(* IEC 61131-3 sources: TA/Tests/RetainTest/Man (part 6) *)

    RETAINTEST_AUTO_ARRAYARRAY_TIME[1][0] := RETAINTEST_AUTO_ARRAYARRAY_TIME[1][0] + PULSE_TIME;
    RETAINTEST_AUTO_ARRAYARRAY_TIME[1][1] := RETAINTEST_AUTO_ARRAYARRAY_TIME[1][1] + PULSE_TIME;
    RETAINTEST_AUTO_ARRAYARRAY_TIME[1][2] := RETAINTEST_AUTO_ARRAYARRAY_TIME[1][2] + PULSE_TIME;
    RETAINTEST_AUTO_ARRAYARRAY_TIME[1][3] := RETAINTEST_AUTO_ARRAYARRAY_TIME[1][3] + PULSE_TIME;
    RETAINTEST_AUTO_ARRAYARRAY_TIME[1][4] := RETAINTEST_AUTO_ARRAYARRAY_TIME[1][4] + PULSE_TIME;
    RETAINTEST_AUTO_ARRAYARRAY_TIME[1][5] := RETAINTEST_AUTO_ARRAYARRAY_TIME[1][5] + PULSE_TIME;
    RETAINTEST_AUTO_ARRAYARRAY_TIME[1][6] := RETAINTEST_AUTO_ARRAYARRAY_TIME[1][6] + PULSE_TIME;
    RETAINTEST_AUTO_ARRAYARRAY_TIME[1][7] := RETAINTEST_AUTO_ARRAYARRAY_TIME[1][7] + PULSE_TIME;
    RETAINTEST_AUTO_ARRAYARRAY_TIME[1][8] := RETAINTEST_AUTO_ARRAYARRAY_TIME[1][6];
    RETAINTEST_AUTO_ARRAYARRAY_TIME[1][9] := RETAINTEST_AUTO_ARRAYARRAY_TIME[1][7];

    RETAINTEST_AUTO_ARRAYARRAY_TIME[2][0] := RETAINTEST_AUTO_ARRAYARRAY_TIME[2][0] + PULSE_TIME;
    RETAINTEST_AUTO_ARRAYARRAY_TIME[2][1] := RETAINTEST_AUTO_ARRAYARRAY_TIME[2][1] + PULSE_TIME;
    RETAINTEST_AUTO_ARRAYARRAY_TIME[2][2] := RETAINTEST_AUTO_ARRAYARRAY_TIME[2][2] + PULSE_TIME;
    RETAINTEST_AUTO_ARRAYARRAY_TIME[2][3] := RETAINTEST_AUTO_ARRAYARRAY_TIME[2][3] + PULSE_TIME;
    RETAINTEST_AUTO_ARRAYARRAY_TIME[2][4] := RETAINTEST_AUTO_ARRAYARRAY_TIME[2][4] + PULSE_TIME;
    RETAINTEST_AUTO_ARRAYARRAY_TIME[2][5] := RETAINTEST_AUTO_ARRAYARRAY_TIME[2][5] + PULSE_TIME;
    RETAINTEST_AUTO_ARRAYARRAY_TIME[2][6] := RETAINTEST_AUTO_ARRAYARRAY_TIME[2][6] + PULSE_TIME;
    RETAINTEST_AUTO_ARRAYARRAY_TIME[2][7] := RETAINTEST_AUTO_ARRAYARRAY_TIME[2][7] + PULSE_TIME;
    RETAINTEST_AUTO_ARRAYARRAY_TIME[2][8] := RETAINTEST_AUTO_ARRAYARRAY_TIME[2][8] + PULSE_TIME;
    RETAINTEST_AUTO_ARRAYARRAY_TIME[2][9] := RETAINTEST_AUTO_ARRAYARRAY_TIME[2][9] + PULSE_TIME;

    RETAINTEST_AUTO_ARRAYARRAY_TIME[3][0] := RETAINTEST_AUTO_ARRAYARRAY_TIME[3][0] + PULSE_TIME;
    RETAINTEST_AUTO_ARRAYARRAY_TIME[3][1] := RETAINTEST_AUTO_ARRAYARRAY_TIME[3][1] + PULSE_TIME;
    RETAINTEST_AUTO_ARRAYARRAY_TIME[3][2] := RETAINTEST_AUTO_ARRAYARRAY_TIME[3][2] + PULSE_TIME;
    RETAINTEST_AUTO_ARRAYARRAY_TIME[3][3] := RETAINTEST_AUTO_ARRAYARRAY_TIME[3][3] + PULSE_TIME;
    RETAINTEST_AUTO_ARRAYARRAY_TIME[3][4] := RETAINTEST_AUTO_ARRAYARRAY_TIME[3][4] + PULSE_TIME;
    RETAINTEST_AUTO_ARRAYARRAY_TIME[3][5] := RETAINTEST_AUTO_ARRAYARRAY_TIME[3][5] + PULSE_TIME;
    RETAINTEST_AUTO_ARRAYARRAY_TIME[3][6] := RETAINTEST_AUTO_ARRAYARRAY_TIME[3][6] + PULSE_TIME;
    RETAINTEST_AUTO_ARRAYARRAY_TIME[3][7] := RETAINTEST_AUTO_ARRAYARRAY_TIME[3][7] + PULSE_TIME;
    RETAINTEST_AUTO_ARRAYARRAY_TIME[3][8] := RETAINTEST_AUTO_ARRAYARRAY_TIME[3][8] + PULSE_TIME;
    RETAINTEST_AUTO_ARRAYARRAY_TIME[3][9] := RETAINTEST_AUTO_ARRAYARRAY_TIME[3][9] + PULSE_TIME;

    RETAINTEST_AUTO_ARRAYARRAY_TIME[4][0] := RETAINTEST_AUTO_ARRAYARRAY_TIME[4][0] + PULSE_TIME;
    RETAINTEST_AUTO_ARRAYARRAY_TIME[4][1] := RETAINTEST_AUTO_ARRAYARRAY_TIME[4][1] + PULSE_TIME;
    RETAINTEST_AUTO_ARRAYARRAY_TIME[4][2] := RETAINTEST_AUTO_ARRAYARRAY_TIME[4][2] + PULSE_TIME;
    RETAINTEST_AUTO_ARRAYARRAY_TIME[4][3] := RETAINTEST_AUTO_ARRAYARRAY_TIME[4][3] + PULSE_TIME;
    RETAINTEST_AUTO_ARRAYARRAY_TIME[4][4] := RETAINTEST_AUTO_ARRAYARRAY_TIME[4][4] + PULSE_TIME;
    RETAINTEST_AUTO_ARRAYARRAY_TIME[4][5] := RETAINTEST_AUTO_ARRAYARRAY_TIME[4][5] + PULSE_TIME;
    RETAINTEST_AUTO_ARRAYARRAY_TIME[4][6] := RETAINTEST_AUTO_ARRAYARRAY_TIME[4][6] + PULSE_TIME;
    RETAINTEST_AUTO_ARRAYARRAY_TIME[4][7] := RETAINTEST_AUTO_ARRAYARRAY_TIME[4][7] + PULSE_TIME;
    RETAINTEST_AUTO_ARRAYARRAY_TIME[4][8] := RETAINTEST_AUTO_ARRAYARRAY_TIME[4][8] + PULSE_TIME;
    RETAINTEST_AUTO_ARRAYARRAY_TIME[4][9] := RETAINTEST_AUTO_ARRAYARRAY_TIME[4][9] + PULSE_TIME;

    RETAINTEST_AUTO_ARRAYARRAY_TIME[5][0] := RETAINTEST_AUTO_ARRAYARRAY_TIME[5][0] + PULSE_TIME;
    RETAINTEST_AUTO_ARRAYARRAY_TIME[5][1] := RETAINTEST_AUTO_ARRAYARRAY_TIME[5][1] + PULSE_TIME;
    RETAINTEST_AUTO_ARRAYARRAY_TIME[5][2] := RETAINTEST_AUTO_ARRAYARRAY_TIME[5][2] + PULSE_TIME;
    RETAINTEST_AUTO_ARRAYARRAY_TIME[5][3] := RETAINTEST_AUTO_ARRAYARRAY_TIME[5][3] + PULSE_TIME;
    RETAINTEST_AUTO_ARRAYARRAY_TIME[5][4] := RETAINTEST_AUTO_ARRAYARRAY_TIME[5][4] + PULSE_TIME;
    RETAINTEST_AUTO_ARRAYARRAY_TIME[5][5] := RETAINTEST_AUTO_ARRAYARRAY_TIME[5][5] + PULSE_TIME;
    RETAINTEST_AUTO_ARRAYARRAY_TIME[5][6] := RETAINTEST_AUTO_ARRAYARRAY_TIME[5][6] + PULSE_TIME;
    RETAINTEST_AUTO_ARRAYARRAY_TIME[5][7] := RETAINTEST_AUTO_ARRAYARRAY_TIME[5][7] + PULSE_TIME;
    RETAINTEST_AUTO_ARRAYARRAY_TIME[5][8] := RETAINTEST_AUTO_ARRAYARRAY_TIME[5][8] + PULSE_TIME;
    RETAINTEST_AUTO_ARRAYARRAY_TIME[5][9] := RETAINTEST_AUTO_ARRAYARRAY_TIME[5][9] + PULSE_TIME;

    RETAINTEST_AUTO_ARRAYARRAY_TIME[6][0] := RETAINTEST_AUTO_ARRAYARRAY_TIME[6][0] + PULSE_TIME;
    RETAINTEST_AUTO_ARRAYARRAY_TIME[6][1] := RETAINTEST_AUTO_ARRAYARRAY_TIME[6][1] + PULSE_TIME;
    RETAINTEST_AUTO_ARRAYARRAY_TIME[6][2] := RETAINTEST_AUTO_ARRAYARRAY_TIME[6][2] + PULSE_TIME;
    RETAINTEST_AUTO_ARRAYARRAY_TIME[6][3] := RETAINTEST_AUTO_ARRAYARRAY_TIME[6][3] + PULSE_TIME;
    RETAINTEST_AUTO_ARRAYARRAY_TIME[6][4] := RETAINTEST_AUTO_ARRAYARRAY_TIME[6][4] + PULSE_TIME;
    RETAINTEST_AUTO_ARRAYARRAY_TIME[6][5] := RETAINTEST_AUTO_ARRAYARRAY_TIME[6][5] + PULSE_TIME;
    RETAINTEST_AUTO_ARRAYARRAY_TIME[6][6] := RETAINTEST_AUTO_ARRAYARRAY_TIME[6][6] + PULSE_TIME;
    RETAINTEST_AUTO_ARRAYARRAY_TIME[6][7] := RETAINTEST_AUTO_ARRAYARRAY_TIME[6][7] + PULSE_TIME;
    RETAINTEST_AUTO_ARRAYARRAY_TIME[6][8] := RETAINTEST_AUTO_ARRAYARRAY_TIME[6][8] + PULSE_TIME;
    RETAINTEST_AUTO_ARRAYARRAY_TIME[6][9] := RETAINTEST_AUTO_ARRAYARRAY_TIME[6][9] + PULSE_TIME;

    RETAINTEST_AUTO_ARRAYARRAY_TIME[7][0] := RETAINTEST_AUTO_ARRAYARRAY_TIME[6][0];
    RETAINTEST_AUTO_ARRAYARRAY_TIME[7][1] := RETAINTEST_AUTO_ARRAYARRAY_TIME[6][1];
    RETAINTEST_AUTO_ARRAYARRAY_TIME[7][2] := RETAINTEST_AUTO_ARRAYARRAY_TIME[6][2];
    RETAINTEST_AUTO_ARRAYARRAY_TIME[7][3] := RETAINTEST_AUTO_ARRAYARRAY_TIME[6][3];
    RETAINTEST_AUTO_ARRAYARRAY_TIME[7][4] := RETAINTEST_AUTO_ARRAYARRAY_TIME[6][4];
    RETAINTEST_AUTO_ARRAYARRAY_TIME[7][5] := RETAINTEST_AUTO_ARRAYARRAY_TIME[6][5];
    RETAINTEST_AUTO_ARRAYARRAY_TIME[7][6] := RETAINTEST_AUTO_ARRAYARRAY_TIME[6][6];
    RETAINTEST_AUTO_ARRAYARRAY_TIME[7][7] := RETAINTEST_AUTO_ARRAYARRAY_TIME[6][7];
    RETAINTEST_AUTO_ARRAYARRAY_TIME[7][8] := RETAINTEST_AUTO_ARRAYARRAY_TIME[6][8];
    RETAINTEST_AUTO_ARRAYARRAY_TIME[7][9] := RETAINTEST_AUTO_ARRAYARRAY_TIME[6][9];

    RETAINTEST_AUTO_ARRAYARRAY_UDINT[0][0] := RETAINTEST_AUTO_ARRAYARRAY_UDINT[0][0] + 1;
    RETAINTEST_AUTO_ARRAYARRAY_UDINT[0][1] := RETAINTEST_AUTO_ARRAYARRAY_UDINT[0][1] + 1;
    RETAINTEST_AUTO_ARRAYARRAY_UDINT[0][2] := RETAINTEST_AUTO_ARRAYARRAY_UDINT[0][2] + 1;
    RETAINTEST_AUTO_ARRAYARRAY_UDINT[0][3] := RETAINTEST_AUTO_ARRAYARRAY_UDINT[0][3] + 1;
    RETAINTEST_AUTO_ARRAYARRAY_UDINT[0][4] := RETAINTEST_AUTO_ARRAYARRAY_UDINT[0][4] + 1;
    RETAINTEST_AUTO_ARRAYARRAY_UDINT[0][5] := RETAINTEST_AUTO_ARRAYARRAY_UDINT[0][5] + 1;
    RETAINTEST_AUTO_ARRAYARRAY_UDINT[0][6] := RETAINTEST_AUTO_ARRAYARRAY_UDINT[0][6] + 1;
    RETAINTEST_AUTO_ARRAYARRAY_UDINT[0][7] := RETAINTEST_AUTO_ARRAYARRAY_UDINT[0][7] + 1;
    RETAINTEST_AUTO_ARRAYARRAY_UDINT[0][8] := RETAINTEST_AUTO_ARRAYARRAY_UDINT[0][6];
    RETAINTEST_AUTO_ARRAYARRAY_UDINT[0][9] := RETAINTEST_AUTO_ARRAYARRAY_UDINT[0][7];

    RETAINTEST_AUTO_ARRAYARRAY_UDINT[1][0] := RETAINTEST_AUTO_ARRAYARRAY_UDINT[1][0] + 1;
    RETAINTEST_AUTO_ARRAYARRAY_UDINT[1][1] := RETAINTEST_AUTO_ARRAYARRAY_UDINT[1][1] + 1;
    RETAINTEST_AUTO_ARRAYARRAY_UDINT[1][2] := RETAINTEST_AUTO_ARRAYARRAY_UDINT[1][2] + 1;
    RETAINTEST_AUTO_ARRAYARRAY_UDINT[1][3] := RETAINTEST_AUTO_ARRAYARRAY_UDINT[1][3] + 1;
    RETAINTEST_AUTO_ARRAYARRAY_UDINT[1][4] := RETAINTEST_AUTO_ARRAYARRAY_UDINT[1][4] + 1;
    RETAINTEST_AUTO_ARRAYARRAY_UDINT[1][5] := RETAINTEST_AUTO_ARRAYARRAY_UDINT[1][5] + 1;
    RETAINTEST_AUTO_ARRAYARRAY_UDINT[1][6] := RETAINTEST_AUTO_ARRAYARRAY_UDINT[1][6] + 1;
    RETAINTEST_AUTO_ARRAYARRAY_UDINT[1][7] := RETAINTEST_AUTO_ARRAYARRAY_UDINT[1][7] + 1;
    RETAINTEST_AUTO_ARRAYARRAY_UDINT[1][8] := RETAINTEST_AUTO_ARRAYARRAY_UDINT[1][6];
    RETAINTEST_AUTO_ARRAYARRAY_UDINT[1][9] := RETAINTEST_AUTO_ARRAYARRAY_UDINT[1][7];

    RETAINTEST_AUTO_ARRAYARRAY_UDINT[2][0] := RETAINTEST_AUTO_ARRAYARRAY_UDINT[2][0] + 1;
    RETAINTEST_AUTO_ARRAYARRAY_UDINT[2][1] := RETAINTEST_AUTO_ARRAYARRAY_UDINT[2][1] + 1;
    RETAINTEST_AUTO_ARRAYARRAY_UDINT[2][2] := RETAINTEST_AUTO_ARRAYARRAY_UDINT[2][2] + 1;
    RETAINTEST_AUTO_ARRAYARRAY_UDINT[2][3] := RETAINTEST_AUTO_ARRAYARRAY_UDINT[2][3] + 1;
    RETAINTEST_AUTO_ARRAYARRAY_UDINT[2][4] := RETAINTEST_AUTO_ARRAYARRAY_UDINT[2][4] + 1;
    RETAINTEST_AUTO_ARRAYARRAY_UDINT[2][5] := RETAINTEST_AUTO_ARRAYARRAY_UDINT[2][5] + 1;
    RETAINTEST_AUTO_ARRAYARRAY_UDINT[2][6] := RETAINTEST_AUTO_ARRAYARRAY_UDINT[2][6] + 1;
    RETAINTEST_AUTO_ARRAYARRAY_UDINT[2][7] := RETAINTEST_AUTO_ARRAYARRAY_UDINT[2][7] + 1;
    RETAINTEST_AUTO_ARRAYARRAY_UDINT[2][8] := RETAINTEST_AUTO_ARRAYARRAY_UDINT[2][8] + 1;
    RETAINTEST_AUTO_ARRAYARRAY_UDINT[2][9] := RETAINTEST_AUTO_ARRAYARRAY_UDINT[2][9] + 1;

    RETAINTEST_AUTO_ARRAYARRAY_UDINT[3][0] := RETAINTEST_AUTO_ARRAYARRAY_UDINT[3][0] + 1;
    RETAINTEST_AUTO_ARRAYARRAY_UDINT[3][1] := RETAINTEST_AUTO_ARRAYARRAY_UDINT[3][1] + 1;
    RETAINTEST_AUTO_ARRAYARRAY_UDINT[3][2] := RETAINTEST_AUTO_ARRAYARRAY_UDINT[3][2] + 1;
    RETAINTEST_AUTO_ARRAYARRAY_UDINT[3][3] := RETAINTEST_AUTO_ARRAYARRAY_UDINT[3][3] + 1;
    RETAINTEST_AUTO_ARRAYARRAY_UDINT[3][4] := RETAINTEST_AUTO_ARRAYARRAY_UDINT[3][4] + 1;
    RETAINTEST_AUTO_ARRAYARRAY_UDINT[3][5] := RETAINTEST_AUTO_ARRAYARRAY_UDINT[3][5] + 1;
    RETAINTEST_AUTO_ARRAYARRAY_UDINT[3][6] := RETAINTEST_AUTO_ARRAYARRAY_UDINT[3][6] + 1;
    RETAINTEST_AUTO_ARRAYARRAY_UDINT[3][7] := RETAINTEST_AUTO_ARRAYARRAY_UDINT[3][7] + 1;
    RETAINTEST_AUTO_ARRAYARRAY_UDINT[3][8] := RETAINTEST_AUTO_ARRAYARRAY_UDINT[3][8] + 1;
    RETAINTEST_AUTO_ARRAYARRAY_UDINT[3][9] := RETAINTEST_AUTO_ARRAYARRAY_UDINT[3][9] + 1;

    RETAINTEST_AUTO_ARRAYARRAY_UDINT[4][0] := RETAINTEST_AUTO_ARRAYARRAY_UDINT[4][0] + 1;
    RETAINTEST_AUTO_ARRAYARRAY_UDINT[4][1] := RETAINTEST_AUTO_ARRAYARRAY_UDINT[4][1] + 1;
    RETAINTEST_AUTO_ARRAYARRAY_UDINT[4][2] := RETAINTEST_AUTO_ARRAYARRAY_UDINT[4][2] + 1;
    RETAINTEST_AUTO_ARRAYARRAY_UDINT[4][3] := RETAINTEST_AUTO_ARRAYARRAY_UDINT[4][3] + 1;
    RETAINTEST_AUTO_ARRAYARRAY_UDINT[4][4] := RETAINTEST_AUTO_ARRAYARRAY_UDINT[4][4] + 1;
    RETAINTEST_AUTO_ARRAYARRAY_UDINT[4][5] := RETAINTEST_AUTO_ARRAYARRAY_UDINT[4][5] + 1;
    RETAINTEST_AUTO_ARRAYARRAY_UDINT[4][6] := RETAINTEST_AUTO_ARRAYARRAY_UDINT[4][6] + 1;
    RETAINTEST_AUTO_ARRAYARRAY_UDINT[4][7] := RETAINTEST_AUTO_ARRAYARRAY_UDINT[4][7] + 1;
    RETAINTEST_AUTO_ARRAYARRAY_UDINT[4][8] := RETAINTEST_AUTO_ARRAYARRAY_UDINT[4][8] + 1;
    RETAINTEST_AUTO_ARRAYARRAY_UDINT[4][9] := RETAINTEST_AUTO_ARRAYARRAY_UDINT[4][9] + 1;

    RETAINTEST_AUTO_ARRAYARRAY_UDINT[5][0] := RETAINTEST_AUTO_ARRAYARRAY_UDINT[5][0] + 1;
    RETAINTEST_AUTO_ARRAYARRAY_UDINT[5][1] := RETAINTEST_AUTO_ARRAYARRAY_UDINT[5][1] + 1;
    RETAINTEST_AUTO_ARRAYARRAY_UDINT[5][2] := RETAINTEST_AUTO_ARRAYARRAY_UDINT[5][2] + 1;
    RETAINTEST_AUTO_ARRAYARRAY_UDINT[5][3] := RETAINTEST_AUTO_ARRAYARRAY_UDINT[5][3] + 1;
    RETAINTEST_AUTO_ARRAYARRAY_UDINT[5][4] := RETAINTEST_AUTO_ARRAYARRAY_UDINT[5][4] + 1;
    RETAINTEST_AUTO_ARRAYARRAY_UDINT[5][5] := RETAINTEST_AUTO_ARRAYARRAY_UDINT[5][5] + 1;
    RETAINTEST_AUTO_ARRAYARRAY_UDINT[5][6] := RETAINTEST_AUTO_ARRAYARRAY_UDINT[5][6] + 1;
    RETAINTEST_AUTO_ARRAYARRAY_UDINT[5][7] := RETAINTEST_AUTO_ARRAYARRAY_UDINT[5][7] + 1;
    RETAINTEST_AUTO_ARRAYARRAY_UDINT[5][8] := RETAINTEST_AUTO_ARRAYARRAY_UDINT[5][8] + 1;
    RETAINTEST_AUTO_ARRAYARRAY_UDINT[5][9] := RETAINTEST_AUTO_ARRAYARRAY_UDINT[5][9] + 1;

    RETAINTEST_AUTO_ARRAYARRAY_UDINT[6][0] := RETAINTEST_AUTO_ARRAYARRAY_UDINT[6][0] + 1;
    RETAINTEST_AUTO_ARRAYARRAY_UDINT[6][1] := RETAINTEST_AUTO_ARRAYARRAY_UDINT[6][1] + 1;
    RETAINTEST_AUTO_ARRAYARRAY_UDINT[6][2] := RETAINTEST_AUTO_ARRAYARRAY_UDINT[6][2] + 1;
    RETAINTEST_AUTO_ARRAYARRAY_UDINT[6][3] := RETAINTEST_AUTO_ARRAYARRAY_UDINT[6][3] + 1;
    RETAINTEST_AUTO_ARRAYARRAY_UDINT[6][4] := RETAINTEST_AUTO_ARRAYARRAY_UDINT[6][4] + 1;
    RETAINTEST_AUTO_ARRAYARRAY_UDINT[6][5] := RETAINTEST_AUTO_ARRAYARRAY_UDINT[6][5] + 1;
    RETAINTEST_AUTO_ARRAYARRAY_UDINT[6][6] := RETAINTEST_AUTO_ARRAYARRAY_UDINT[6][6] + 1;
    RETAINTEST_AUTO_ARRAYARRAY_UDINT[6][7] := RETAINTEST_AUTO_ARRAYARRAY_UDINT[6][7] + 1;
    RETAINTEST_AUTO_ARRAYARRAY_UDINT[6][8] := RETAINTEST_AUTO_ARRAYARRAY_UDINT[6][8] + 1;
    RETAINTEST_AUTO_ARRAYARRAY_UDINT[6][9] := RETAINTEST_AUTO_ARRAYARRAY_UDINT[6][9] + 1;

    RETAINTEST_AUTO_ARRAYARRAY_UDINT[7][0] := RETAINTEST_AUTO_ARRAYARRAY_UDINT[6][0];
    RETAINTEST_AUTO_ARRAYARRAY_UDINT[7][1] := RETAINTEST_AUTO_ARRAYARRAY_UDINT[6][1];
    RETAINTEST_AUTO_ARRAYARRAY_UDINT[7][2] := RETAINTEST_AUTO_ARRAYARRAY_UDINT[6][2];
    RETAINTEST_AUTO_ARRAYARRAY_UDINT[7][3] := RETAINTEST_AUTO_ARRAYARRAY_UDINT[6][3];
    RETAINTEST_AUTO_ARRAYARRAY_UDINT[7][4] := RETAINTEST_AUTO_ARRAYARRAY_UDINT[6][4];
    RETAINTEST_AUTO_ARRAYARRAY_UDINT[7][5] := RETAINTEST_AUTO_ARRAYARRAY_UDINT[6][5];
    RETAINTEST_AUTO_ARRAYARRAY_UDINT[7][6] := RETAINTEST_AUTO_ARRAYARRAY_UDINT[6][6];
    RETAINTEST_AUTO_ARRAYARRAY_UDINT[7][7] := RETAINTEST_AUTO_ARRAYARRAY_UDINT[6][7];
    RETAINTEST_AUTO_ARRAYARRAY_UDINT[7][8] := RETAINTEST_AUTO_ARRAYARRAY_UDINT[6][8];
    RETAINTEST_AUTO_ARRAYARRAY_UDINT[7][9] := RETAINTEST_AUTO_ARRAYARRAY_UDINT[6][9];

    RETAINTEST_AUTO_ARRAYARRAY_UINT[0][0] := RETAINTEST_AUTO_ARRAYARRAY_UINT[0][0] + 1;
    RETAINTEST_AUTO_ARRAYARRAY_UINT[0][1] := RETAINTEST_AUTO_ARRAYARRAY_UINT[0][1] + 1;
    RETAINTEST_AUTO_ARRAYARRAY_UINT[0][2] := RETAINTEST_AUTO_ARRAYARRAY_UINT[0][2] + 1;
    RETAINTEST_AUTO_ARRAYARRAY_UINT[0][3] := RETAINTEST_AUTO_ARRAYARRAY_UINT[0][3] + 1;
    RETAINTEST_AUTO_ARRAYARRAY_UINT[0][4] := RETAINTEST_AUTO_ARRAYARRAY_UINT[0][4] + 1;
    RETAINTEST_AUTO_ARRAYARRAY_UINT[0][5] := RETAINTEST_AUTO_ARRAYARRAY_UINT[0][5] + 1;
    RETAINTEST_AUTO_ARRAYARRAY_UINT[0][6] := RETAINTEST_AUTO_ARRAYARRAY_UINT[0][6] + 1;
    RETAINTEST_AUTO_ARRAYARRAY_UINT[0][7] := RETAINTEST_AUTO_ARRAYARRAY_UINT[0][7] + 1;
    RETAINTEST_AUTO_ARRAYARRAY_UINT[0][8] := RETAINTEST_AUTO_ARRAYARRAY_UINT[0][6];
    RETAINTEST_AUTO_ARRAYARRAY_UINT[0][9] := RETAINTEST_AUTO_ARRAYARRAY_UINT[0][7];

    RETAINTEST_AUTO_ARRAYARRAY_UINT[1][0] := RETAINTEST_AUTO_ARRAYARRAY_UINT[1][0] + 1;
    RETAINTEST_AUTO_ARRAYARRAY_UINT[1][1] := RETAINTEST_AUTO_ARRAYARRAY_UINT[1][1] + 1;
    RETAINTEST_AUTO_ARRAYARRAY_UINT[1][2] := RETAINTEST_AUTO_ARRAYARRAY_UINT[1][2] + 1;
    RETAINTEST_AUTO_ARRAYARRAY_UINT[1][3] := RETAINTEST_AUTO_ARRAYARRAY_UINT[1][3] + 1;
    RETAINTEST_AUTO_ARRAYARRAY_UINT[1][4] := RETAINTEST_AUTO_ARRAYARRAY_UINT[1][4] + 1;
    RETAINTEST_AUTO_ARRAYARRAY_UINT[1][5] := RETAINTEST_AUTO_ARRAYARRAY_UINT[1][5] + 1;
    RETAINTEST_AUTO_ARRAYARRAY_UINT[1][6] := RETAINTEST_AUTO_ARRAYARRAY_UINT[1][6] + 1;
    RETAINTEST_AUTO_ARRAYARRAY_UINT[1][7] := RETAINTEST_AUTO_ARRAYARRAY_UINT[1][7] + 1;
    RETAINTEST_AUTO_ARRAYARRAY_UINT[1][8] := RETAINTEST_AUTO_ARRAYARRAY_UINT[1][6];
    RETAINTEST_AUTO_ARRAYARRAY_UINT[1][9] := RETAINTEST_AUTO_ARRAYARRAY_UINT[1][7];

    RETAINTEST_AUTO_ARRAYARRAY_UINT[2][0] := RETAINTEST_AUTO_ARRAYARRAY_UINT[2][0] + 1;
    RETAINTEST_AUTO_ARRAYARRAY_UINT[2][1] := RETAINTEST_AUTO_ARRAYARRAY_UINT[2][1] + 1;
    RETAINTEST_AUTO_ARRAYARRAY_UINT[2][2] := RETAINTEST_AUTO_ARRAYARRAY_UINT[2][2] + 1;
    RETAINTEST_AUTO_ARRAYARRAY_UINT[2][3] := RETAINTEST_AUTO_ARRAYARRAY_UINT[2][3] + 1;
    RETAINTEST_AUTO_ARRAYARRAY_UINT[2][4] := RETAINTEST_AUTO_ARRAYARRAY_UINT[2][4] + 1;
    RETAINTEST_AUTO_ARRAYARRAY_UINT[2][5] := RETAINTEST_AUTO_ARRAYARRAY_UINT[2][5] + 1;
    RETAINTEST_AUTO_ARRAYARRAY_UINT[2][6] := RETAINTEST_AUTO_ARRAYARRAY_UINT[2][6] + 1;
    RETAINTEST_AUTO_ARRAYARRAY_UINT[2][7] := RETAINTEST_AUTO_ARRAYARRAY_UINT[2][7] + 1;
    RETAINTEST_AUTO_ARRAYARRAY_UINT[2][8] := RETAINTEST_AUTO_ARRAYARRAY_UINT[2][8] + 1;
    RETAINTEST_AUTO_ARRAYARRAY_UINT[2][9] := RETAINTEST_AUTO_ARRAYARRAY_UINT[2][9] + 1;

    RETAINTEST_AUTO_ARRAYARRAY_UINT[3][0] := RETAINTEST_AUTO_ARRAYARRAY_UINT[3][0] + 1;
    RETAINTEST_AUTO_ARRAYARRAY_UINT[3][1] := RETAINTEST_AUTO_ARRAYARRAY_UINT[3][1] + 1;
    RETAINTEST_AUTO_ARRAYARRAY_UINT[3][2] := RETAINTEST_AUTO_ARRAYARRAY_UINT[3][2] + 1;
    RETAINTEST_AUTO_ARRAYARRAY_UINT[3][3] := RETAINTEST_AUTO_ARRAYARRAY_UINT[3][3] + 1;
    RETAINTEST_AUTO_ARRAYARRAY_UINT[3][4] := RETAINTEST_AUTO_ARRAYARRAY_UINT[3][4] + 1;
    RETAINTEST_AUTO_ARRAYARRAY_UINT[3][5] := RETAINTEST_AUTO_ARRAYARRAY_UINT[3][5] + 1;
    RETAINTEST_AUTO_ARRAYARRAY_UINT[3][6] := RETAINTEST_AUTO_ARRAYARRAY_UINT[3][6] + 1;
    RETAINTEST_AUTO_ARRAYARRAY_UINT[3][7] := RETAINTEST_AUTO_ARRAYARRAY_UINT[3][7] + 1;
    RETAINTEST_AUTO_ARRAYARRAY_UINT[3][8] := RETAINTEST_AUTO_ARRAYARRAY_UINT[3][8] + 1;
    RETAINTEST_AUTO_ARRAYARRAY_UINT[3][9] := RETAINTEST_AUTO_ARRAYARRAY_UINT[3][9] + 1;

    RETAINTEST_AUTO_ARRAYARRAY_UINT[4][0] := RETAINTEST_AUTO_ARRAYARRAY_UINT[4][0] + 1;
    RETAINTEST_AUTO_ARRAYARRAY_UINT[4][1] := RETAINTEST_AUTO_ARRAYARRAY_UINT[4][1] + 1;
    RETAINTEST_AUTO_ARRAYARRAY_UINT[4][2] := RETAINTEST_AUTO_ARRAYARRAY_UINT[4][2] + 1;
    RETAINTEST_AUTO_ARRAYARRAY_UINT[4][3] := RETAINTEST_AUTO_ARRAYARRAY_UINT[4][3] + 1;
    RETAINTEST_AUTO_ARRAYARRAY_UINT[4][4] := RETAINTEST_AUTO_ARRAYARRAY_UINT[4][4] + 1;
    RETAINTEST_AUTO_ARRAYARRAY_UINT[4][5] := RETAINTEST_AUTO_ARRAYARRAY_UINT[4][5] + 1;
    RETAINTEST_AUTO_ARRAYARRAY_UINT[4][6] := RETAINTEST_AUTO_ARRAYARRAY_UINT[4][6] + 1;
    RETAINTEST_AUTO_ARRAYARRAY_UINT[4][7] := RETAINTEST_AUTO_ARRAYARRAY_UINT[4][7] + 1;
    RETAINTEST_AUTO_ARRAYARRAY_UINT[4][8] := RETAINTEST_AUTO_ARRAYARRAY_UINT[4][8] + 1;
    RETAINTEST_AUTO_ARRAYARRAY_UINT[4][9] := RETAINTEST_AUTO_ARRAYARRAY_UINT[4][9] + 1;

    RETAINTEST_AUTO_ARRAYARRAY_UINT[5][0] := RETAINTEST_AUTO_ARRAYARRAY_UINT[5][0] + 1;
    RETAINTEST_AUTO_ARRAYARRAY_UINT[5][1] := RETAINTEST_AUTO_ARRAYARRAY_UINT[5][1] + 1;
    RETAINTEST_AUTO_ARRAYARRAY_UINT[5][2] := RETAINTEST_AUTO_ARRAYARRAY_UINT[5][2] + 1;
    RETAINTEST_AUTO_ARRAYARRAY_UINT[5][3] := RETAINTEST_AUTO_ARRAYARRAY_UINT[5][3] + 1;
    RETAINTEST_AUTO_ARRAYARRAY_UINT[5][4] := RETAINTEST_AUTO_ARRAYARRAY_UINT[5][4] + 1;
    RETAINTEST_AUTO_ARRAYARRAY_UINT[5][5] := RETAINTEST_AUTO_ARRAYARRAY_UINT[5][5] + 1;
    RETAINTEST_AUTO_ARRAYARRAY_UINT[5][6] := RETAINTEST_AUTO_ARRAYARRAY_UINT[5][6] + 1;
    RETAINTEST_AUTO_ARRAYARRAY_UINT[5][7] := RETAINTEST_AUTO_ARRAYARRAY_UINT[5][7] + 1;
    RETAINTEST_AUTO_ARRAYARRAY_UINT[5][8] := RETAINTEST_AUTO_ARRAYARRAY_UINT[5][8] + 1;
    RETAINTEST_AUTO_ARRAYARRAY_UINT[5][9] := RETAINTEST_AUTO_ARRAYARRAY_UINT[5][9] + 1;

    RETAINTEST_AUTO_ARRAYARRAY_UINT[6][0] := RETAINTEST_AUTO_ARRAYARRAY_UINT[6][0] + 1;
    RETAINTEST_AUTO_ARRAYARRAY_UINT[6][1] := RETAINTEST_AUTO_ARRAYARRAY_UINT[6][1] + 1;
    RETAINTEST_AUTO_ARRAYARRAY_UINT[6][2] := RETAINTEST_AUTO_ARRAYARRAY_UINT[6][2] + 1;
    RETAINTEST_AUTO_ARRAYARRAY_UINT[6][3] := RETAINTEST_AUTO_ARRAYARRAY_UINT[6][3] + 1;
    RETAINTEST_AUTO_ARRAYARRAY_UINT[6][4] := RETAINTEST_AUTO_ARRAYARRAY_UINT[6][4] + 1;
    RETAINTEST_AUTO_ARRAYARRAY_UINT[6][5] := RETAINTEST_AUTO_ARRAYARRAY_UINT[6][5] + 1;
    RETAINTEST_AUTO_ARRAYARRAY_UINT[6][6] := RETAINTEST_AUTO_ARRAYARRAY_UINT[6][6] + 1;
    RETAINTEST_AUTO_ARRAYARRAY_UINT[6][7] := RETAINTEST_AUTO_ARRAYARRAY_UINT[6][7] + 1;
    RETAINTEST_AUTO_ARRAYARRAY_UINT[6][8] := RETAINTEST_AUTO_ARRAYARRAY_UINT[6][8] + 1;
    RETAINTEST_AUTO_ARRAYARRAY_UINT[6][9] := RETAINTEST_AUTO_ARRAYARRAY_UINT[6][9] + 1;

    RETAINTEST_AUTO_ARRAYARRAY_UINT[7][0] := RETAINTEST_AUTO_ARRAYARRAY_UINT[6][0];
    RETAINTEST_AUTO_ARRAYARRAY_UINT[7][1] := RETAINTEST_AUTO_ARRAYARRAY_UINT[6][1];
    RETAINTEST_AUTO_ARRAYARRAY_UINT[7][2] := RETAINTEST_AUTO_ARRAYARRAY_UINT[6][2];
    RETAINTEST_AUTO_ARRAYARRAY_UINT[7][3] := RETAINTEST_AUTO_ARRAYARRAY_UINT[6][3];
    RETAINTEST_AUTO_ARRAYARRAY_UINT[7][4] := RETAINTEST_AUTO_ARRAYARRAY_UINT[6][4];
    RETAINTEST_AUTO_ARRAYARRAY_UINT[7][5] := RETAINTEST_AUTO_ARRAYARRAY_UINT[6][5];
    RETAINTEST_AUTO_ARRAYARRAY_UINT[7][6] := RETAINTEST_AUTO_ARRAYARRAY_UINT[6][6];
    RETAINTEST_AUTO_ARRAYARRAY_UINT[7][7] := RETAINTEST_AUTO_ARRAYARRAY_UINT[6][7];
    RETAINTEST_AUTO_ARRAYARRAY_UINT[7][8] := RETAINTEST_AUTO_ARRAYARRAY_UINT[6][8];
    RETAINTEST_AUTO_ARRAYARRAY_UINT[7][9] := RETAINTEST_AUTO_ARRAYARRAY_UINT[6][9];

    RETAINTEST_AUTO_ARRAYARRAY_ULINT[0][0] := RETAINTEST_AUTO_ARRAYARRAY_ULINT[0][0] + 1;
    RETAINTEST_AUTO_ARRAYARRAY_ULINT[0][1] := RETAINTEST_AUTO_ARRAYARRAY_ULINT[0][1] + 1;
    RETAINTEST_AUTO_ARRAYARRAY_ULINT[0][2] := RETAINTEST_AUTO_ARRAYARRAY_ULINT[0][2] + 1;
    RETAINTEST_AUTO_ARRAYARRAY_ULINT[0][3] := RETAINTEST_AUTO_ARRAYARRAY_ULINT[0][3] + 1;
    RETAINTEST_AUTO_ARRAYARRAY_ULINT[0][4] := RETAINTEST_AUTO_ARRAYARRAY_ULINT[0][4] + 1;
    RETAINTEST_AUTO_ARRAYARRAY_ULINT[0][5] := RETAINTEST_AUTO_ARRAYARRAY_ULINT[0][5] + 1;
    RETAINTEST_AUTO_ARRAYARRAY_ULINT[0][6] := RETAINTEST_AUTO_ARRAYARRAY_ULINT[0][6] + 1;
    RETAINTEST_AUTO_ARRAYARRAY_ULINT[0][7] := RETAINTEST_AUTO_ARRAYARRAY_ULINT[0][7] + 1;
    RETAINTEST_AUTO_ARRAYARRAY_ULINT[0][8] := RETAINTEST_AUTO_ARRAYARRAY_ULINT[0][6];
    RETAINTEST_AUTO_ARRAYARRAY_ULINT[0][9] := RETAINTEST_AUTO_ARRAYARRAY_ULINT[0][7];

    RETAINTEST_AUTO_ARRAYARRAY_ULINT[1][0] := RETAINTEST_AUTO_ARRAYARRAY_ULINT[1][0] + 1;
    RETAINTEST_AUTO_ARRAYARRAY_ULINT[1][1] := RETAINTEST_AUTO_ARRAYARRAY_ULINT[1][1] + 1;
    RETAINTEST_AUTO_ARRAYARRAY_ULINT[1][2] := RETAINTEST_AUTO_ARRAYARRAY_ULINT[1][2] + 1;
    RETAINTEST_AUTO_ARRAYARRAY_ULINT[1][3] := RETAINTEST_AUTO_ARRAYARRAY_ULINT[1][3] + 1;
    RETAINTEST_AUTO_ARRAYARRAY_ULINT[1][4] := RETAINTEST_AUTO_ARRAYARRAY_ULINT[1][4] + 1;
    RETAINTEST_AUTO_ARRAYARRAY_ULINT[1][5] := RETAINTEST_AUTO_ARRAYARRAY_ULINT[1][5] + 1;
    RETAINTEST_AUTO_ARRAYARRAY_ULINT[1][6] := RETAINTEST_AUTO_ARRAYARRAY_ULINT[1][6] + 1;
    RETAINTEST_AUTO_ARRAYARRAY_ULINT[1][7] := RETAINTEST_AUTO_ARRAYARRAY_ULINT[1][7] + 1;
    RETAINTEST_AUTO_ARRAYARRAY_ULINT[1][8] := RETAINTEST_AUTO_ARRAYARRAY_ULINT[1][6];
    RETAINTEST_AUTO_ARRAYARRAY_ULINT[1][9] := RETAINTEST_AUTO_ARRAYARRAY_ULINT[1][7];

    RETAINTEST_AUTO_ARRAYARRAY_ULINT[2][0] := RETAINTEST_AUTO_ARRAYARRAY_ULINT[2][0] + 1;
    RETAINTEST_AUTO_ARRAYARRAY_ULINT[2][1] := RETAINTEST_AUTO_ARRAYARRAY_ULINT[2][1] + 1;
    RETAINTEST_AUTO_ARRAYARRAY_ULINT[2][2] := RETAINTEST_AUTO_ARRAYARRAY_ULINT[2][2] + 1;
    RETAINTEST_AUTO_ARRAYARRAY_ULINT[2][3] := RETAINTEST_AUTO_ARRAYARRAY_ULINT[2][3] + 1;
    RETAINTEST_AUTO_ARRAYARRAY_ULINT[2][4] := RETAINTEST_AUTO_ARRAYARRAY_ULINT[2][4] + 1;
    RETAINTEST_AUTO_ARRAYARRAY_ULINT[2][5] := RETAINTEST_AUTO_ARRAYARRAY_ULINT[2][5] + 1;
    RETAINTEST_AUTO_ARRAYARRAY_ULINT[2][6] := RETAINTEST_AUTO_ARRAYARRAY_ULINT[2][6] + 1;
    RETAINTEST_AUTO_ARRAYARRAY_ULINT[2][7] := RETAINTEST_AUTO_ARRAYARRAY_ULINT[2][7] + 1;
    RETAINTEST_AUTO_ARRAYARRAY_ULINT[2][8] := RETAINTEST_AUTO_ARRAYARRAY_ULINT[2][8] + 1;
    RETAINTEST_AUTO_ARRAYARRAY_ULINT[2][9] := RETAINTEST_AUTO_ARRAYARRAY_ULINT[2][9] + 1;

    RETAINTEST_AUTO_ARRAYARRAY_ULINT[3][0] := RETAINTEST_AUTO_ARRAYARRAY_ULINT[3][0] + 1;
    RETAINTEST_AUTO_ARRAYARRAY_ULINT[3][1] := RETAINTEST_AUTO_ARRAYARRAY_ULINT[3][1] + 1;
    RETAINTEST_AUTO_ARRAYARRAY_ULINT[3][2] := RETAINTEST_AUTO_ARRAYARRAY_ULINT[3][2] + 1;
    RETAINTEST_AUTO_ARRAYARRAY_ULINT[3][3] := RETAINTEST_AUTO_ARRAYARRAY_ULINT[3][3] + 1;
    RETAINTEST_AUTO_ARRAYARRAY_ULINT[3][4] := RETAINTEST_AUTO_ARRAYARRAY_ULINT[3][4] + 1;
    RETAINTEST_AUTO_ARRAYARRAY_ULINT[3][5] := RETAINTEST_AUTO_ARRAYARRAY_ULINT[3][5] + 1;
    RETAINTEST_AUTO_ARRAYARRAY_ULINT[3][6] := RETAINTEST_AUTO_ARRAYARRAY_ULINT[3][6] + 1;
    RETAINTEST_AUTO_ARRAYARRAY_ULINT[3][7] := RETAINTEST_AUTO_ARRAYARRAY_ULINT[3][7] + 1;
    RETAINTEST_AUTO_ARRAYARRAY_ULINT[3][8] := RETAINTEST_AUTO_ARRAYARRAY_ULINT[3][8] + 1;
    RETAINTEST_AUTO_ARRAYARRAY_ULINT[3][9] := RETAINTEST_AUTO_ARRAYARRAY_ULINT[3][9] + 1;

    RETAINTEST_AUTO_ARRAYARRAY_ULINT[4][0] := RETAINTEST_AUTO_ARRAYARRAY_ULINT[4][0] + 1;
    RETAINTEST_AUTO_ARRAYARRAY_ULINT[4][1] := RETAINTEST_AUTO_ARRAYARRAY_ULINT[4][1] + 1;
    RETAINTEST_AUTO_ARRAYARRAY_ULINT[4][2] := RETAINTEST_AUTO_ARRAYARRAY_ULINT[4][2] + 1;
    RETAINTEST_AUTO_ARRAYARRAY_ULINT[4][3] := RETAINTEST_AUTO_ARRAYARRAY_ULINT[4][3] + 1;
    RETAINTEST_AUTO_ARRAYARRAY_ULINT[4][4] := RETAINTEST_AUTO_ARRAYARRAY_ULINT[4][4] + 1;
    RETAINTEST_AUTO_ARRAYARRAY_ULINT[4][5] := RETAINTEST_AUTO_ARRAYARRAY_ULINT[4][5] + 1;
    RETAINTEST_AUTO_ARRAYARRAY_ULINT[4][6] := RETAINTEST_AUTO_ARRAYARRAY_ULINT[4][6] + 1;
    RETAINTEST_AUTO_ARRAYARRAY_ULINT[4][7] := RETAINTEST_AUTO_ARRAYARRAY_ULINT[4][7] + 1;
    RETAINTEST_AUTO_ARRAYARRAY_ULINT[4][8] := RETAINTEST_AUTO_ARRAYARRAY_ULINT[4][8] + 1;
    RETAINTEST_AUTO_ARRAYARRAY_ULINT[4][9] := RETAINTEST_AUTO_ARRAYARRAY_ULINT[4][9] + 1;

    RETAINTEST_AUTO_ARRAYARRAY_ULINT[5][0] := RETAINTEST_AUTO_ARRAYARRAY_ULINT[5][0] + 1;
    RETAINTEST_AUTO_ARRAYARRAY_ULINT[5][1] := RETAINTEST_AUTO_ARRAYARRAY_ULINT[5][1] + 1;
    RETAINTEST_AUTO_ARRAYARRAY_ULINT[5][2] := RETAINTEST_AUTO_ARRAYARRAY_ULINT[5][2] + 1;
    RETAINTEST_AUTO_ARRAYARRAY_ULINT[5][3] := RETAINTEST_AUTO_ARRAYARRAY_ULINT[5][3] + 1;
    RETAINTEST_AUTO_ARRAYARRAY_ULINT[5][4] := RETAINTEST_AUTO_ARRAYARRAY_ULINT[5][4] + 1;
    RETAINTEST_AUTO_ARRAYARRAY_ULINT[5][5] := RETAINTEST_AUTO_ARRAYARRAY_ULINT[5][5] + 1;
    RETAINTEST_AUTO_ARRAYARRAY_ULINT[5][6] := RETAINTEST_AUTO_ARRAYARRAY_ULINT[5][6] + 1;
    RETAINTEST_AUTO_ARRAYARRAY_ULINT[5][7] := RETAINTEST_AUTO_ARRAYARRAY_ULINT[5][7] + 1;
    RETAINTEST_AUTO_ARRAYARRAY_ULINT[5][8] := RETAINTEST_AUTO_ARRAYARRAY_ULINT[5][8] + 1;
    RETAINTEST_AUTO_ARRAYARRAY_ULINT[5][9] := RETAINTEST_AUTO_ARRAYARRAY_ULINT[5][9] + 1;

    RETAINTEST_AUTO_ARRAYARRAY_ULINT[6][0] := RETAINTEST_AUTO_ARRAYARRAY_ULINT[6][0] + 1;
    RETAINTEST_AUTO_ARRAYARRAY_ULINT[6][1] := RETAINTEST_AUTO_ARRAYARRAY_ULINT[6][1] + 1;
    RETAINTEST_AUTO_ARRAYARRAY_ULINT[6][2] := RETAINTEST_AUTO_ARRAYARRAY_ULINT[6][2] + 1;
    RETAINTEST_AUTO_ARRAYARRAY_ULINT[6][3] := RETAINTEST_AUTO_ARRAYARRAY_ULINT[6][3] + 1;
    RETAINTEST_AUTO_ARRAYARRAY_ULINT[6][4] := RETAINTEST_AUTO_ARRAYARRAY_ULINT[6][4] + 1;
    RETAINTEST_AUTO_ARRAYARRAY_ULINT[6][5] := RETAINTEST_AUTO_ARRAYARRAY_ULINT[6][5] + 1;
    RETAINTEST_AUTO_ARRAYARRAY_ULINT[6][6] := RETAINTEST_AUTO_ARRAYARRAY_ULINT[6][6] + 1;
    RETAINTEST_AUTO_ARRAYARRAY_ULINT[6][7] := RETAINTEST_AUTO_ARRAYARRAY_ULINT[6][7] + 1;
    RETAINTEST_AUTO_ARRAYARRAY_ULINT[6][8] := RETAINTEST_AUTO_ARRAYARRAY_ULINT[6][8] + 1;
    RETAINTEST_AUTO_ARRAYARRAY_ULINT[6][9] := RETAINTEST_AUTO_ARRAYARRAY_ULINT[6][9] + 1;

    RETAINTEST_AUTO_ARRAYARRAY_ULINT[7][0] := RETAINTEST_AUTO_ARRAYARRAY_ULINT[6][0];
    RETAINTEST_AUTO_ARRAYARRAY_ULINT[7][1] := RETAINTEST_AUTO_ARRAYARRAY_ULINT[6][1];
    RETAINTEST_AUTO_ARRAYARRAY_ULINT[7][2] := RETAINTEST_AUTO_ARRAYARRAY_ULINT[6][2];
    RETAINTEST_AUTO_ARRAYARRAY_ULINT[7][3] := RETAINTEST_AUTO_ARRAYARRAY_ULINT[6][3];
    RETAINTEST_AUTO_ARRAYARRAY_ULINT[7][4] := RETAINTEST_AUTO_ARRAYARRAY_ULINT[6][4];
    RETAINTEST_AUTO_ARRAYARRAY_ULINT[7][5] := RETAINTEST_AUTO_ARRAYARRAY_ULINT[6][5];
    RETAINTEST_AUTO_ARRAYARRAY_ULINT[7][6] := RETAINTEST_AUTO_ARRAYARRAY_ULINT[6][6];
    RETAINTEST_AUTO_ARRAYARRAY_ULINT[7][7] := RETAINTEST_AUTO_ARRAYARRAY_ULINT[6][7];
    RETAINTEST_AUTO_ARRAYARRAY_ULINT[7][8] := RETAINTEST_AUTO_ARRAYARRAY_ULINT[6][8];
    RETAINTEST_AUTO_ARRAYARRAY_ULINT[7][9] := RETAINTEST_AUTO_ARRAYARRAY_ULINT[6][9];

    RETAINTEST_AUTO_ARRAYARRAY_USINT[0][0] := RETAINTEST_AUTO_ARRAYARRAY_USINT[0][0] + 1;
    RETAINTEST_AUTO_ARRAYARRAY_USINT[0][1] := RETAINTEST_AUTO_ARRAYARRAY_USINT[0][1] + 1;
    RETAINTEST_AUTO_ARRAYARRAY_USINT[0][2] := RETAINTEST_AUTO_ARRAYARRAY_USINT[0][2] + 1;
    RETAINTEST_AUTO_ARRAYARRAY_USINT[0][3] := RETAINTEST_AUTO_ARRAYARRAY_USINT[0][3] + 1;
    RETAINTEST_AUTO_ARRAYARRAY_USINT[0][4] := RETAINTEST_AUTO_ARRAYARRAY_USINT[0][4] + 1;
    RETAINTEST_AUTO_ARRAYARRAY_USINT[0][5] := RETAINTEST_AUTO_ARRAYARRAY_USINT[0][5] + 1;
    RETAINTEST_AUTO_ARRAYARRAY_USINT[0][6] := RETAINTEST_AUTO_ARRAYARRAY_USINT[0][6] + 1;
    RETAINTEST_AUTO_ARRAYARRAY_USINT[0][7] := RETAINTEST_AUTO_ARRAYARRAY_USINT[0][7] + 1;
    RETAINTEST_AUTO_ARRAYARRAY_USINT[0][8] := RETAINTEST_AUTO_ARRAYARRAY_USINT[0][6];
    RETAINTEST_AUTO_ARRAYARRAY_USINT[0][9] := RETAINTEST_AUTO_ARRAYARRAY_USINT[0][7];

    RETAINTEST_AUTO_ARRAYARRAY_USINT[1][0] := RETAINTEST_AUTO_ARRAYARRAY_USINT[1][0] + 1;
    RETAINTEST_AUTO_ARRAYARRAY_USINT[1][1] := RETAINTEST_AUTO_ARRAYARRAY_USINT[1][1] + 1;
    RETAINTEST_AUTO_ARRAYARRAY_USINT[1][2] := RETAINTEST_AUTO_ARRAYARRAY_USINT[1][2] + 1;
    RETAINTEST_AUTO_ARRAYARRAY_USINT[1][3] := RETAINTEST_AUTO_ARRAYARRAY_USINT[1][3] + 1;
    RETAINTEST_AUTO_ARRAYARRAY_USINT[1][4] := RETAINTEST_AUTO_ARRAYARRAY_USINT[1][4] + 1;
    RETAINTEST_AUTO_ARRAYARRAY_USINT[1][5] := RETAINTEST_AUTO_ARRAYARRAY_USINT[1][5] + 1;
    RETAINTEST_AUTO_ARRAYARRAY_USINT[1][6] := RETAINTEST_AUTO_ARRAYARRAY_USINT[1][6] + 1;
    RETAINTEST_AUTO_ARRAYARRAY_USINT[1][7] := RETAINTEST_AUTO_ARRAYARRAY_USINT[1][7] + 1;
    RETAINTEST_AUTO_ARRAYARRAY_USINT[1][8] := RETAINTEST_AUTO_ARRAYARRAY_USINT[1][6];
    RETAINTEST_AUTO_ARRAYARRAY_USINT[1][9] := RETAINTEST_AUTO_ARRAYARRAY_USINT[1][7];

    RETAINTEST_AUTO_ARRAYARRAY_USINT[2][0] := RETAINTEST_AUTO_ARRAYARRAY_USINT[2][0] + 1;
    RETAINTEST_AUTO_ARRAYARRAY_USINT[2][1] := RETAINTEST_AUTO_ARRAYARRAY_USINT[2][1] + 1;
    RETAINTEST_AUTO_ARRAYARRAY_USINT[2][2] := RETAINTEST_AUTO_ARRAYARRAY_USINT[2][2] + 1;
    RETAINTEST_AUTO_ARRAYARRAY_USINT[2][3] := RETAINTEST_AUTO_ARRAYARRAY_USINT[2][3] + 1;
    RETAINTEST_AUTO_ARRAYARRAY_USINT[2][4] := RETAINTEST_AUTO_ARRAYARRAY_USINT[2][4] + 1;
    RETAINTEST_AUTO_ARRAYARRAY_USINT[2][5] := RETAINTEST_AUTO_ARRAYARRAY_USINT[2][5] + 1;
    RETAINTEST_AUTO_ARRAYARRAY_USINT[2][6] := RETAINTEST_AUTO_ARRAYARRAY_USINT[2][6] + 1;
    RETAINTEST_AUTO_ARRAYARRAY_USINT[2][7] := RETAINTEST_AUTO_ARRAYARRAY_USINT[2][7] + 1;
    RETAINTEST_AUTO_ARRAYARRAY_USINT[2][8] := RETAINTEST_AUTO_ARRAYARRAY_USINT[2][8] + 1;
    RETAINTEST_AUTO_ARRAYARRAY_USINT[2][9] := RETAINTEST_AUTO_ARRAYARRAY_USINT[2][9] + 1;

    RETAINTEST_AUTO_ARRAYARRAY_USINT[3][0] := RETAINTEST_AUTO_ARRAYARRAY_USINT[3][0] + 1;
    RETAINTEST_AUTO_ARRAYARRAY_USINT[3][1] := RETAINTEST_AUTO_ARRAYARRAY_USINT[3][1] + 1;
    RETAINTEST_AUTO_ARRAYARRAY_USINT[3][2] := RETAINTEST_AUTO_ARRAYARRAY_USINT[3][2] + 1;
    RETAINTEST_AUTO_ARRAYARRAY_USINT[3][3] := RETAINTEST_AUTO_ARRAYARRAY_USINT[3][3] + 1;
    RETAINTEST_AUTO_ARRAYARRAY_USINT[3][4] := RETAINTEST_AUTO_ARRAYARRAY_USINT[3][4] + 1;
    RETAINTEST_AUTO_ARRAYARRAY_USINT[3][5] := RETAINTEST_AUTO_ARRAYARRAY_USINT[3][5] + 1;
    RETAINTEST_AUTO_ARRAYARRAY_USINT[3][6] := RETAINTEST_AUTO_ARRAYARRAY_USINT[3][6] + 1;
    RETAINTEST_AUTO_ARRAYARRAY_USINT[3][7] := RETAINTEST_AUTO_ARRAYARRAY_USINT[3][7] + 1;
    RETAINTEST_AUTO_ARRAYARRAY_USINT[3][8] := RETAINTEST_AUTO_ARRAYARRAY_USINT[3][8] + 1;
    RETAINTEST_AUTO_ARRAYARRAY_USINT[3][9] := RETAINTEST_AUTO_ARRAYARRAY_USINT[3][9] + 1;

    RETAINTEST_AUTO_ARRAYARRAY_USINT[4][0] := RETAINTEST_AUTO_ARRAYARRAY_USINT[4][0] + 1;
    RETAINTEST_AUTO_ARRAYARRAY_USINT[4][1] := RETAINTEST_AUTO_ARRAYARRAY_USINT[4][1] + 1;
    RETAINTEST_AUTO_ARRAYARRAY_USINT[4][2] := RETAINTEST_AUTO_ARRAYARRAY_USINT[4][2] + 1;
    RETAINTEST_AUTO_ARRAYARRAY_USINT[4][3] := RETAINTEST_AUTO_ARRAYARRAY_USINT[4][3] + 1;
    RETAINTEST_AUTO_ARRAYARRAY_USINT[4][4] := RETAINTEST_AUTO_ARRAYARRAY_USINT[4][4] + 1;
    RETAINTEST_AUTO_ARRAYARRAY_USINT[4][5] := RETAINTEST_AUTO_ARRAYARRAY_USINT[4][5] + 1;
    RETAINTEST_AUTO_ARRAYARRAY_USINT[4][6] := RETAINTEST_AUTO_ARRAYARRAY_USINT[4][6] + 1;
    RETAINTEST_AUTO_ARRAYARRAY_USINT[4][7] := RETAINTEST_AUTO_ARRAYARRAY_USINT[4][7] + 1;
    RETAINTEST_AUTO_ARRAYARRAY_USINT[4][8] := RETAINTEST_AUTO_ARRAYARRAY_USINT[4][8] + 1;
    RETAINTEST_AUTO_ARRAYARRAY_USINT[4][9] := RETAINTEST_AUTO_ARRAYARRAY_USINT[4][9] + 1;

    RETAINTEST_AUTO_ARRAYARRAY_USINT[5][0] := RETAINTEST_AUTO_ARRAYARRAY_USINT[5][0] + 1;
    RETAINTEST_AUTO_ARRAYARRAY_USINT[5][1] := RETAINTEST_AUTO_ARRAYARRAY_USINT[5][1] + 1;
    RETAINTEST_AUTO_ARRAYARRAY_USINT[5][2] := RETAINTEST_AUTO_ARRAYARRAY_USINT[5][2] + 1;
    RETAINTEST_AUTO_ARRAYARRAY_USINT[5][3] := RETAINTEST_AUTO_ARRAYARRAY_USINT[5][3] + 1;
    RETAINTEST_AUTO_ARRAYARRAY_USINT[5][4] := RETAINTEST_AUTO_ARRAYARRAY_USINT[5][4] + 1;
    RETAINTEST_AUTO_ARRAYARRAY_USINT[5][5] := RETAINTEST_AUTO_ARRAYARRAY_USINT[5][5] + 1;
    RETAINTEST_AUTO_ARRAYARRAY_USINT[5][6] := RETAINTEST_AUTO_ARRAYARRAY_USINT[5][6] + 1;
    RETAINTEST_AUTO_ARRAYARRAY_USINT[5][7] := RETAINTEST_AUTO_ARRAYARRAY_USINT[5][7] + 1;
    RETAINTEST_AUTO_ARRAYARRAY_USINT[5][8] := RETAINTEST_AUTO_ARRAYARRAY_USINT[5][8] + 1;
    RETAINTEST_AUTO_ARRAYARRAY_USINT[5][9] := RETAINTEST_AUTO_ARRAYARRAY_USINT[5][9] + 1;

    RETAINTEST_AUTO_ARRAYARRAY_USINT[6][0] := RETAINTEST_AUTO_ARRAYARRAY_USINT[6][0] + 1;
    RETAINTEST_AUTO_ARRAYARRAY_USINT[6][1] := RETAINTEST_AUTO_ARRAYARRAY_USINT[6][1] + 1;
    RETAINTEST_AUTO_ARRAYARRAY_USINT[6][2] := RETAINTEST_AUTO_ARRAYARRAY_USINT[6][2] + 1;
    RETAINTEST_AUTO_ARRAYARRAY_USINT[6][3] := RETAINTEST_AUTO_ARRAYARRAY_USINT[6][3] + 1;
    RETAINTEST_AUTO_ARRAYARRAY_USINT[6][4] := RETAINTEST_AUTO_ARRAYARRAY_USINT[6][4] + 1;
    RETAINTEST_AUTO_ARRAYARRAY_USINT[6][5] := RETAINTEST_AUTO_ARRAYARRAY_USINT[6][5] + 1;
    RETAINTEST_AUTO_ARRAYARRAY_USINT[6][6] := RETAINTEST_AUTO_ARRAYARRAY_USINT[6][6] + 1;
    RETAINTEST_AUTO_ARRAYARRAY_USINT[6][7] := RETAINTEST_AUTO_ARRAYARRAY_USINT[6][7] + 1;
    RETAINTEST_AUTO_ARRAYARRAY_USINT[6][8] := RETAINTEST_AUTO_ARRAYARRAY_USINT[6][8] + 1;
    RETAINTEST_AUTO_ARRAYARRAY_USINT[6][9] := RETAINTEST_AUTO_ARRAYARRAY_USINT[6][9] + 1;

    RETAINTEST_AUTO_ARRAYARRAY_USINT[7][0] := RETAINTEST_AUTO_ARRAYARRAY_USINT[6][0];
    RETAINTEST_AUTO_ARRAYARRAY_USINT[7][1] := RETAINTEST_AUTO_ARRAYARRAY_USINT[6][1];
    RETAINTEST_AUTO_ARRAYARRAY_USINT[7][2] := RETAINTEST_AUTO_ARRAYARRAY_USINT[6][2];
    RETAINTEST_AUTO_ARRAYARRAY_USINT[7][3] := RETAINTEST_AUTO_ARRAYARRAY_USINT[6][3];
    RETAINTEST_AUTO_ARRAYARRAY_USINT[7][4] := RETAINTEST_AUTO_ARRAYARRAY_USINT[6][4];
    RETAINTEST_AUTO_ARRAYARRAY_USINT[7][5] := RETAINTEST_AUTO_ARRAYARRAY_USINT[6][5];
    RETAINTEST_AUTO_ARRAYARRAY_USINT[7][6] := RETAINTEST_AUTO_ARRAYARRAY_USINT[6][6];
    RETAINTEST_AUTO_ARRAYARRAY_USINT[7][7] := RETAINTEST_AUTO_ARRAYARRAY_USINT[6][7];
    RETAINTEST_AUTO_ARRAYARRAY_USINT[7][8] := RETAINTEST_AUTO_ARRAYARRAY_USINT[6][8];
    RETAINTEST_AUTO_ARRAYARRAY_USINT[7][9] := RETAINTEST_AUTO_ARRAYARRAY_USINT[6][9];

    RETAINTEST_AUTO_ARRAYARRAY_WORD[0][0] := RETAINTEST_AUTO_ARRAYARRAY_WORD[0][0] + 1;
    RETAINTEST_AUTO_ARRAYARRAY_WORD[0][1] := RETAINTEST_AUTO_ARRAYARRAY_WORD[0][1] + 1;
    RETAINTEST_AUTO_ARRAYARRAY_WORD[0][2] := RETAINTEST_AUTO_ARRAYARRAY_WORD[0][2] + 1;
    RETAINTEST_AUTO_ARRAYARRAY_WORD[0][3] := RETAINTEST_AUTO_ARRAYARRAY_WORD[0][3] + 1;
    RETAINTEST_AUTO_ARRAYARRAY_WORD[0][4] := RETAINTEST_AUTO_ARRAYARRAY_WORD[0][4] + 1;
    RETAINTEST_AUTO_ARRAYARRAY_WORD[0][5] := RETAINTEST_AUTO_ARRAYARRAY_WORD[0][5] + 1;
    RETAINTEST_AUTO_ARRAYARRAY_WORD[0][6] := RETAINTEST_AUTO_ARRAYARRAY_WORD[0][6] + 1;
    RETAINTEST_AUTO_ARRAYARRAY_WORD[0][7] := RETAINTEST_AUTO_ARRAYARRAY_WORD[0][7] + 1;
    RETAINTEST_AUTO_ARRAYARRAY_WORD[0][8] := RETAINTEST_AUTO_ARRAYARRAY_WORD[0][6];
    RETAINTEST_AUTO_ARRAYARRAY_WORD[0][9] := RETAINTEST_AUTO_ARRAYARRAY_WORD[0][7];

    RETAINTEST_AUTO_ARRAYARRAY_WORD[1][0] := RETAINTEST_AUTO_ARRAYARRAY_WORD[1][0] + 1;
    RETAINTEST_AUTO_ARRAYARRAY_WORD[1][1] := RETAINTEST_AUTO_ARRAYARRAY_WORD[1][1] + 1;
    RETAINTEST_AUTO_ARRAYARRAY_WORD[1][2] := RETAINTEST_AUTO_ARRAYARRAY_WORD[1][2] + 1;
    RETAINTEST_AUTO_ARRAYARRAY_WORD[1][3] := RETAINTEST_AUTO_ARRAYARRAY_WORD[1][3] + 1;
    RETAINTEST_AUTO_ARRAYARRAY_WORD[1][4] := RETAINTEST_AUTO_ARRAYARRAY_WORD[1][4] + 1;
    RETAINTEST_AUTO_ARRAYARRAY_WORD[1][5] := RETAINTEST_AUTO_ARRAYARRAY_WORD[1][5] + 1;
    RETAINTEST_AUTO_ARRAYARRAY_WORD[1][6] := RETAINTEST_AUTO_ARRAYARRAY_WORD[1][6] + 1;
    RETAINTEST_AUTO_ARRAYARRAY_WORD[1][7] := RETAINTEST_AUTO_ARRAYARRAY_WORD[1][7] + 1;
    RETAINTEST_AUTO_ARRAYARRAY_WORD[1][8] := RETAINTEST_AUTO_ARRAYARRAY_WORD[1][6];
    RETAINTEST_AUTO_ARRAYARRAY_WORD[1][9] := RETAINTEST_AUTO_ARRAYARRAY_WORD[1][7];

    RETAINTEST_AUTO_ARRAYARRAY_WORD[2][0] := RETAINTEST_AUTO_ARRAYARRAY_WORD[2][0] + 1;
    RETAINTEST_AUTO_ARRAYARRAY_WORD[2][1] := RETAINTEST_AUTO_ARRAYARRAY_WORD[2][1] + 1;
    RETAINTEST_AUTO_ARRAYARRAY_WORD[2][2] := RETAINTEST_AUTO_ARRAYARRAY_WORD[2][2] + 1;
    RETAINTEST_AUTO_ARRAYARRAY_WORD[2][3] := RETAINTEST_AUTO_ARRAYARRAY_WORD[2][3] + 1;
    RETAINTEST_AUTO_ARRAYARRAY_WORD[2][4] := RETAINTEST_AUTO_ARRAYARRAY_WORD[2][4] + 1;
    RETAINTEST_AUTO_ARRAYARRAY_WORD[2][5] := RETAINTEST_AUTO_ARRAYARRAY_WORD[2][5] + 1;
    RETAINTEST_AUTO_ARRAYARRAY_WORD[2][6] := RETAINTEST_AUTO_ARRAYARRAY_WORD[2][6] + 1;
    RETAINTEST_AUTO_ARRAYARRAY_WORD[2][7] := RETAINTEST_AUTO_ARRAYARRAY_WORD[2][7] + 1;
    RETAINTEST_AUTO_ARRAYARRAY_WORD[2][8] := RETAINTEST_AUTO_ARRAYARRAY_WORD[2][8] + 1;
    RETAINTEST_AUTO_ARRAYARRAY_WORD[2][9] := RETAINTEST_AUTO_ARRAYARRAY_WORD[2][9] + 1;

    RETAINTEST_AUTO_ARRAYARRAY_WORD[3][0] := RETAINTEST_AUTO_ARRAYARRAY_WORD[3][0] + 1;
    RETAINTEST_AUTO_ARRAYARRAY_WORD[3][1] := RETAINTEST_AUTO_ARRAYARRAY_WORD[3][1] + 1;
    RETAINTEST_AUTO_ARRAYARRAY_WORD[3][2] := RETAINTEST_AUTO_ARRAYARRAY_WORD[3][2] + 1;
    RETAINTEST_AUTO_ARRAYARRAY_WORD[3][3] := RETAINTEST_AUTO_ARRAYARRAY_WORD[3][3] + 1;
    RETAINTEST_AUTO_ARRAYARRAY_WORD[3][4] := RETAINTEST_AUTO_ARRAYARRAY_WORD[3][4] + 1;
    RETAINTEST_AUTO_ARRAYARRAY_WORD[3][5] := RETAINTEST_AUTO_ARRAYARRAY_WORD[3][5] + 1;
    RETAINTEST_AUTO_ARRAYARRAY_WORD[3][6] := RETAINTEST_AUTO_ARRAYARRAY_WORD[3][6] + 1;
    RETAINTEST_AUTO_ARRAYARRAY_WORD[3][7] := RETAINTEST_AUTO_ARRAYARRAY_WORD[3][7] + 1;
    RETAINTEST_AUTO_ARRAYARRAY_WORD[3][8] := RETAINTEST_AUTO_ARRAYARRAY_WORD[3][8] + 1;
    RETAINTEST_AUTO_ARRAYARRAY_WORD[3][9] := RETAINTEST_AUTO_ARRAYARRAY_WORD[3][9] + 1;

    RETAINTEST_AUTO_ARRAYARRAY_WORD[4][0] := RETAINTEST_AUTO_ARRAYARRAY_WORD[4][0] + 1;
    RETAINTEST_AUTO_ARRAYARRAY_WORD[4][1] := RETAINTEST_AUTO_ARRAYARRAY_WORD[4][1] + 1;
    RETAINTEST_AUTO_ARRAYARRAY_WORD[4][2] := RETAINTEST_AUTO_ARRAYARRAY_WORD[4][2] + 1;
    RETAINTEST_AUTO_ARRAYARRAY_WORD[4][3] := RETAINTEST_AUTO_ARRAYARRAY_WORD[4][3] + 1;
    RETAINTEST_AUTO_ARRAYARRAY_WORD[4][4] := RETAINTEST_AUTO_ARRAYARRAY_WORD[4][4] + 1;
    RETAINTEST_AUTO_ARRAYARRAY_WORD[4][5] := RETAINTEST_AUTO_ARRAYARRAY_WORD[4][5] + 1;
    RETAINTEST_AUTO_ARRAYARRAY_WORD[4][6] := RETAINTEST_AUTO_ARRAYARRAY_WORD[4][6] + 1;
    RETAINTEST_AUTO_ARRAYARRAY_WORD[4][7] := RETAINTEST_AUTO_ARRAYARRAY_WORD[4][7] + 1;
    RETAINTEST_AUTO_ARRAYARRAY_WORD[4][8] := RETAINTEST_AUTO_ARRAYARRAY_WORD[4][8] + 1;
    RETAINTEST_AUTO_ARRAYARRAY_WORD[4][9] := RETAINTEST_AUTO_ARRAYARRAY_WORD[4][9] + 1;

    RETAINTEST_AUTO_ARRAYARRAY_WORD[5][0] := RETAINTEST_AUTO_ARRAYARRAY_WORD[5][0] + 1;
    RETAINTEST_AUTO_ARRAYARRAY_WORD[5][1] := RETAINTEST_AUTO_ARRAYARRAY_WORD[5][1] + 1;
    RETAINTEST_AUTO_ARRAYARRAY_WORD[5][2] := RETAINTEST_AUTO_ARRAYARRAY_WORD[5][2] + 1;
    RETAINTEST_AUTO_ARRAYARRAY_WORD[5][3] := RETAINTEST_AUTO_ARRAYARRAY_WORD[5][3] + 1;
    RETAINTEST_AUTO_ARRAYARRAY_WORD[5][4] := RETAINTEST_AUTO_ARRAYARRAY_WORD[5][4] + 1;
    RETAINTEST_AUTO_ARRAYARRAY_WORD[5][5] := RETAINTEST_AUTO_ARRAYARRAY_WORD[5][5] + 1;
    RETAINTEST_AUTO_ARRAYARRAY_WORD[5][6] := RETAINTEST_AUTO_ARRAYARRAY_WORD[5][6] + 1;
    RETAINTEST_AUTO_ARRAYARRAY_WORD[5][7] := RETAINTEST_AUTO_ARRAYARRAY_WORD[5][7] + 1;
    RETAINTEST_AUTO_ARRAYARRAY_WORD[5][8] := RETAINTEST_AUTO_ARRAYARRAY_WORD[5][8] + 1;
    RETAINTEST_AUTO_ARRAYARRAY_WORD[5][9] := RETAINTEST_AUTO_ARRAYARRAY_WORD[5][9] + 1;

    RETAINTEST_AUTO_ARRAYARRAY_WORD[6][0] := RETAINTEST_AUTO_ARRAYARRAY_WORD[6][0] + 1;
    RETAINTEST_AUTO_ARRAYARRAY_WORD[6][1] := RETAINTEST_AUTO_ARRAYARRAY_WORD[6][1] + 1;
    RETAINTEST_AUTO_ARRAYARRAY_WORD[6][2] := RETAINTEST_AUTO_ARRAYARRAY_WORD[6][2] + 1;
    RETAINTEST_AUTO_ARRAYARRAY_WORD[6][3] := RETAINTEST_AUTO_ARRAYARRAY_WORD[6][3] + 1;
    RETAINTEST_AUTO_ARRAYARRAY_WORD[6][4] := RETAINTEST_AUTO_ARRAYARRAY_WORD[6][4] + 1;
    RETAINTEST_AUTO_ARRAYARRAY_WORD[6][5] := RETAINTEST_AUTO_ARRAYARRAY_WORD[6][5] + 1;
    RETAINTEST_AUTO_ARRAYARRAY_WORD[6][6] := RETAINTEST_AUTO_ARRAYARRAY_WORD[6][6] + 1;
    RETAINTEST_AUTO_ARRAYARRAY_WORD[6][7] := RETAINTEST_AUTO_ARRAYARRAY_WORD[6][7] + 1;
    RETAINTEST_AUTO_ARRAYARRAY_WORD[6][8] := RETAINTEST_AUTO_ARRAYARRAY_WORD[6][8] + 1;
    RETAINTEST_AUTO_ARRAYARRAY_WORD[6][9] := RETAINTEST_AUTO_ARRAYARRAY_WORD[6][9] + 1;

    RETAINTEST_AUTO_ARRAYARRAY_WORD[7][0] := RETAINTEST_AUTO_ARRAYARRAY_WORD[6][0];
    RETAINTEST_AUTO_ARRAYARRAY_WORD[7][1] := RETAINTEST_AUTO_ARRAYARRAY_WORD[6][1];
    RETAINTEST_AUTO_ARRAYARRAY_WORD[7][2] := RETAINTEST_AUTO_ARRAYARRAY_WORD[6][2];
    RETAINTEST_AUTO_ARRAYARRAY_WORD[7][3] := RETAINTEST_AUTO_ARRAYARRAY_WORD[6][3];
    RETAINTEST_AUTO_ARRAYARRAY_WORD[7][4] := RETAINTEST_AUTO_ARRAYARRAY_WORD[6][4];
    RETAINTEST_AUTO_ARRAYARRAY_WORD[7][5] := RETAINTEST_AUTO_ARRAYARRAY_WORD[6][5];
    RETAINTEST_AUTO_ARRAYARRAY_WORD[7][6] := RETAINTEST_AUTO_ARRAYARRAY_WORD[6][6];
    RETAINTEST_AUTO_ARRAYARRAY_WORD[7][7] := RETAINTEST_AUTO_ARRAYARRAY_WORD[6][7];
    RETAINTEST_AUTO_ARRAYARRAY_WORD[7][8] := RETAINTEST_AUTO_ARRAYARRAY_WORD[6][8];
    RETAINTEST_AUTO_ARRAYARRAY_WORD[7][9] := RETAINTEST_AUTO_ARRAYARRAY_WORD[6][9];
END_IF;

END_PROGRAM

(* ---- ManRetainArrayStructureSimple.st ---- *)
PROGRAM ManRetainArrayStructureSimple

IF TRIGGER_IMP.Q AND StartManRetainTest THEN
    RETAINTEST_RETAIN_ARRAYSIMPLESTRUCTURE[0].SIMPLE_BOOL := NOT RETAINTEST_RETAIN_ARRAYSIMPLESTRUCTURE[0].SIMPLE_BOOL;
    RETAINTEST_RETAIN_ARRAYSIMPLESTRUCTURE[0].SIMPLE_BYTE := RETAINTEST_RETAIN_ARRAYSIMPLESTRUCTURE[0].SIMPLE_BYTE + 1;
    RETAINTEST_RETAIN_ARRAYSIMPLESTRUCTURE[0].SIMPLE_DATE := ANY_TO_DATE(1445385600 + RETAINTEST_RETAIN_ARRAYSIMPLESTRUCTURE[0].SIMPLE_DINT * 86400);
    RETAINTEST_RETAIN_ARRAYSIMPLESTRUCTURE[0].SIMPLE_DINT := RETAINTEST_RETAIN_ARRAYSIMPLESTRUCTURE[0].SIMPLE_DINT + 1;
    RETAINTEST_RETAIN_ARRAYSIMPLESTRUCTURE[0].SIMPLE_DWORD := RETAINTEST_RETAIN_ARRAYSIMPLESTRUCTURE[0].SIMPLE_DWORD + 1;
    RETAINTEST_RETAIN_ARRAYSIMPLESTRUCTURE[0].SIMPLE_INT := RETAINTEST_RETAIN_ARRAYSIMPLESTRUCTURE[0].SIMPLE_INT + 1;
    RETAINTEST_RETAIN_ARRAYSIMPLESTRUCTURE[0].SIMPLE_LINT := RETAINTEST_RETAIN_ARRAYSIMPLESTRUCTURE[0].SIMPLE_LINT + 1;
    RETAINTEST_RETAIN_ARRAYSIMPLESTRUCTURE[0].SIMPLE_LREAL := RETAINTEST_RETAIN_ARRAYSIMPLESTRUCTURE[0].SIMPLE_LREAL + 1.1;
    RETAINTEST_RETAIN_ARRAYSIMPLESTRUCTURE[0].SIMPLE_LWORD := RETAINTEST_RETAIN_ARRAYSIMPLESTRUCTURE[0].SIMPLE_LWORD + 1;
    RETAINTEST_RETAIN_ARRAYSIMPLESTRUCTURE[0].SIMPLE_REAL := RETAINTEST_RETAIN_ARRAYSIMPLESTRUCTURE[0].SIMPLE_REAL + 1.1;
    RETAINTEST_RETAIN_ARRAYSIMPLESTRUCTURE[0].SIMPLE_SINT := RETAINTEST_RETAIN_ARRAYSIMPLESTRUCTURE[0].SIMPLE_SINT + 1;
    RETAINTEST_RETAIN_ARRAYSIMPLESTRUCTURE[0].SIMPLE_STRING := ANY_TO_STRING(RETAINTEST_RETAIN_ARRAYSIMPLESTRUCTURE[0].SIMPLE_DINT) + ' ' + ANY_TO_STRING(RETAINTEST_RETAIN_ARRAYSIMPLESTRUCTURE[0].SIMPLE_TIME);
    RETAINTEST_RETAIN_ARRAYSIMPLESTRUCTURE[0].SIMPLE_TIME := RETAINTEST_RETAIN_ARRAYSIMPLESTRUCTURE[0].SIMPLE_TIME + PULSE_TIME;
    RETAINTEST_RETAIN_ARRAYSIMPLESTRUCTURE[0].SIMPLE_UDINT := RETAINTEST_RETAIN_ARRAYSIMPLESTRUCTURE[0].SIMPLE_UDINT + 1;
    RETAINTEST_RETAIN_ARRAYSIMPLESTRUCTURE[0].SIMPLE_UINT := RETAINTEST_RETAIN_ARRAYSIMPLESTRUCTURE[0].SIMPLE_UINT + 1;
    RETAINTEST_RETAIN_ARRAYSIMPLESTRUCTURE[0].SIMPLE_ULINT := RETAINTEST_RETAIN_ARRAYSIMPLESTRUCTURE[0].SIMPLE_ULINT + 1;
    RETAINTEST_RETAIN_ARRAYSIMPLESTRUCTURE[0].SIMPLE_USINT := RETAINTEST_RETAIN_ARRAYSIMPLESTRUCTURE[0].SIMPLE_USINT + 1;
    RETAINTEST_RETAIN_ARRAYSIMPLESTRUCTURE[0].SIMPLE_WORD := RETAINTEST_RETAIN_ARRAYSIMPLESTRUCTURE[0].SIMPLE_WORD + 1;

    RETAINTEST_RETAIN_ARRAYSIMPLESTRUCTURE[1].SIMPLE_BOOL := NOT RETAINTEST_RETAIN_ARRAYSIMPLESTRUCTURE[1].SIMPLE_BOOL;
    RETAINTEST_RETAIN_ARRAYSIMPLESTRUCTURE[1].SIMPLE_BYTE := RETAINTEST_RETAIN_ARRAYSIMPLESTRUCTURE[1].SIMPLE_BYTE + 1;
    RETAINTEST_RETAIN_ARRAYSIMPLESTRUCTURE[1].SIMPLE_DATE := ANY_TO_DATE(1445385600 + RETAINTEST_RETAIN_ARRAYSIMPLESTRUCTURE[1].SIMPLE_DINT * 86400);
    RETAINTEST_RETAIN_ARRAYSIMPLESTRUCTURE[1].SIMPLE_DINT := RETAINTEST_RETAIN_ARRAYSIMPLESTRUCTURE[1].SIMPLE_DINT + 1;
    RETAINTEST_RETAIN_ARRAYSIMPLESTRUCTURE[1].SIMPLE_DWORD := RETAINTEST_RETAIN_ARRAYSIMPLESTRUCTURE[1].SIMPLE_DWORD + 1;
    RETAINTEST_RETAIN_ARRAYSIMPLESTRUCTURE[1].SIMPLE_INT := RETAINTEST_RETAIN_ARRAYSIMPLESTRUCTURE[1].SIMPLE_INT + 1;
    RETAINTEST_RETAIN_ARRAYSIMPLESTRUCTURE[1].SIMPLE_LINT := RETAINTEST_RETAIN_ARRAYSIMPLESTRUCTURE[1].SIMPLE_LINT + 1;
    RETAINTEST_RETAIN_ARRAYSIMPLESTRUCTURE[1].SIMPLE_LREAL := RETAINTEST_RETAIN_ARRAYSIMPLESTRUCTURE[1].SIMPLE_LREAL + 1.1;
    RETAINTEST_RETAIN_ARRAYSIMPLESTRUCTURE[1].SIMPLE_LWORD := RETAINTEST_RETAIN_ARRAYSIMPLESTRUCTURE[1].SIMPLE_LWORD + 1;
    RETAINTEST_RETAIN_ARRAYSIMPLESTRUCTURE[1].SIMPLE_REAL := RETAINTEST_RETAIN_ARRAYSIMPLESTRUCTURE[1].SIMPLE_REAL + 1.1;
    RETAINTEST_RETAIN_ARRAYSIMPLESTRUCTURE[1].SIMPLE_SINT := RETAINTEST_RETAIN_ARRAYSIMPLESTRUCTURE[1].SIMPLE_SINT + 1;
    RETAINTEST_RETAIN_ARRAYSIMPLESTRUCTURE[1].SIMPLE_STRING := ANY_TO_STRING(RETAINTEST_RETAIN_ARRAYSIMPLESTRUCTURE[1].SIMPLE_DINT) + ' ' + ANY_TO_STRING(RETAINTEST_RETAIN_ARRAYSIMPLESTRUCTURE[1].SIMPLE_TIME);
    RETAINTEST_RETAIN_ARRAYSIMPLESTRUCTURE[1].SIMPLE_TIME := RETAINTEST_RETAIN_ARRAYSIMPLESTRUCTURE[1].SIMPLE_TIME + PULSE_TIME;
    RETAINTEST_RETAIN_ARRAYSIMPLESTRUCTURE[1].SIMPLE_UDINT := RETAINTEST_RETAIN_ARRAYSIMPLESTRUCTURE[1].SIMPLE_UDINT + 1;
    RETAINTEST_RETAIN_ARRAYSIMPLESTRUCTURE[1].SIMPLE_UINT := RETAINTEST_RETAIN_ARRAYSIMPLESTRUCTURE[1].SIMPLE_UINT + 1;
    RETAINTEST_RETAIN_ARRAYSIMPLESTRUCTURE[1].SIMPLE_ULINT := RETAINTEST_RETAIN_ARRAYSIMPLESTRUCTURE[1].SIMPLE_ULINT + 1;
    RETAINTEST_RETAIN_ARRAYSIMPLESTRUCTURE[1].SIMPLE_USINT := RETAINTEST_RETAIN_ARRAYSIMPLESTRUCTURE[1].SIMPLE_USINT + 1;
    RETAINTEST_RETAIN_ARRAYSIMPLESTRUCTURE[1].SIMPLE_WORD := RETAINTEST_RETAIN_ARRAYSIMPLESTRUCTURE[1].SIMPLE_WORD + 1;

    RETAINTEST_RETAIN_ARRAYSIMPLESTRUCTURE[2].SIMPLE_BOOL := NOT RETAINTEST_RETAIN_ARRAYSIMPLESTRUCTURE[2].SIMPLE_BOOL;
    RETAINTEST_RETAIN_ARRAYSIMPLESTRUCTURE[2].SIMPLE_BYTE := RETAINTEST_RETAIN_ARRAYSIMPLESTRUCTURE[2].SIMPLE_BYTE + 1;
    RETAINTEST_RETAIN_ARRAYSIMPLESTRUCTURE[2].SIMPLE_DATE := ANY_TO_DATE(1445385600 + RETAINTEST_RETAIN_ARRAYSIMPLESTRUCTURE[2].SIMPLE_DINT * 86400);
    RETAINTEST_RETAIN_ARRAYSIMPLESTRUCTURE[2].SIMPLE_DINT := RETAINTEST_RETAIN_ARRAYSIMPLESTRUCTURE[2].SIMPLE_DINT + 1;
    RETAINTEST_RETAIN_ARRAYSIMPLESTRUCTURE[2].SIMPLE_DWORD := RETAINTEST_RETAIN_ARRAYSIMPLESTRUCTURE[2].SIMPLE_DWORD + 1;
    RETAINTEST_RETAIN_ARRAYSIMPLESTRUCTURE[2].SIMPLE_INT := RETAINTEST_RETAIN_ARRAYSIMPLESTRUCTURE[2].SIMPLE_INT + 1;
    RETAINTEST_RETAIN_ARRAYSIMPLESTRUCTURE[2].SIMPLE_LINT := RETAINTEST_RETAIN_ARRAYSIMPLESTRUCTURE[2].SIMPLE_LINT + 1;
    RETAINTEST_RETAIN_ARRAYSIMPLESTRUCTURE[2].SIMPLE_LREAL := RETAINTEST_RETAIN_ARRAYSIMPLESTRUCTURE[2].SIMPLE_LREAL + 1.1;
    RETAINTEST_RETAIN_ARRAYSIMPLESTRUCTURE[2].SIMPLE_LWORD := RETAINTEST_RETAIN_ARRAYSIMPLESTRUCTURE[2].SIMPLE_LWORD + 1;
    RETAINTEST_RETAIN_ARRAYSIMPLESTRUCTURE[2].SIMPLE_REAL := RETAINTEST_RETAIN_ARRAYSIMPLESTRUCTURE[2].SIMPLE_REAL + 1.1;
    RETAINTEST_RETAIN_ARRAYSIMPLESTRUCTURE[2].SIMPLE_SINT := RETAINTEST_RETAIN_ARRAYSIMPLESTRUCTURE[2].SIMPLE_SINT + 1;
    RETAINTEST_RETAIN_ARRAYSIMPLESTRUCTURE[2].SIMPLE_STRING := ANY_TO_STRING(RETAINTEST_RETAIN_ARRAYSIMPLESTRUCTURE[2].SIMPLE_DINT) + ' ' + ANY_TO_STRING(RETAINTEST_RETAIN_ARRAYSIMPLESTRUCTURE[2].SIMPLE_TIME);
    RETAINTEST_RETAIN_ARRAYSIMPLESTRUCTURE[2].SIMPLE_TIME := RETAINTEST_RETAIN_ARRAYSIMPLESTRUCTURE[2].SIMPLE_TIME + PULSE_TIME;
    RETAINTEST_RETAIN_ARRAYSIMPLESTRUCTURE[2].SIMPLE_UDINT := RETAINTEST_RETAIN_ARRAYSIMPLESTRUCTURE[2].SIMPLE_UDINT + 1;
    RETAINTEST_RETAIN_ARRAYSIMPLESTRUCTURE[2].SIMPLE_UINT := RETAINTEST_RETAIN_ARRAYSIMPLESTRUCTURE[2].SIMPLE_UINT + 1;
    RETAINTEST_RETAIN_ARRAYSIMPLESTRUCTURE[2].SIMPLE_ULINT := RETAINTEST_RETAIN_ARRAYSIMPLESTRUCTURE[2].SIMPLE_ULINT + 1;
    RETAINTEST_RETAIN_ARRAYSIMPLESTRUCTURE[2].SIMPLE_USINT := RETAINTEST_RETAIN_ARRAYSIMPLESTRUCTURE[2].SIMPLE_USINT + 1;
    RETAINTEST_RETAIN_ARRAYSIMPLESTRUCTURE[2].SIMPLE_WORD := RETAINTEST_RETAIN_ARRAYSIMPLESTRUCTURE[2].SIMPLE_WORD + 1;

    RETAINTEST_RETAIN_ARRAYSIMPLESTRUCTURE[3].SIMPLE_BOOL := NOT RETAINTEST_RETAIN_ARRAYSIMPLESTRUCTURE[3].SIMPLE_BOOL;
    RETAINTEST_RETAIN_ARRAYSIMPLESTRUCTURE[3].SIMPLE_BYTE := RETAINTEST_RETAIN_ARRAYSIMPLESTRUCTURE[3].SIMPLE_BYTE + 1;
    RETAINTEST_RETAIN_ARRAYSIMPLESTRUCTURE[3].SIMPLE_DATE := ANY_TO_DATE(1445385600 + RETAINTEST_RETAIN_ARRAYSIMPLESTRUCTURE[3].SIMPLE_DINT * 86400);
    RETAINTEST_RETAIN_ARRAYSIMPLESTRUCTURE[3].SIMPLE_DINT := RETAINTEST_RETAIN_ARRAYSIMPLESTRUCTURE[3].SIMPLE_DINT + 1;
    RETAINTEST_RETAIN_ARRAYSIMPLESTRUCTURE[3].SIMPLE_DWORD := RETAINTEST_RETAIN_ARRAYSIMPLESTRUCTURE[3].SIMPLE_DWORD + 1;
    RETAINTEST_RETAIN_ARRAYSIMPLESTRUCTURE[3].SIMPLE_INT := RETAINTEST_RETAIN_ARRAYSIMPLESTRUCTURE[3].SIMPLE_INT + 1;
    RETAINTEST_RETAIN_ARRAYSIMPLESTRUCTURE[3].SIMPLE_LINT := RETAINTEST_RETAIN_ARRAYSIMPLESTRUCTURE[3].SIMPLE_LINT + 1;
    RETAINTEST_RETAIN_ARRAYSIMPLESTRUCTURE[3].SIMPLE_LREAL := RETAINTEST_RETAIN_ARRAYSIMPLESTRUCTURE[3].SIMPLE_LREAL + 1.1;
    RETAINTEST_RETAIN_ARRAYSIMPLESTRUCTURE[3].SIMPLE_LWORD := RETAINTEST_RETAIN_ARRAYSIMPLESTRUCTURE[3].SIMPLE_LWORD + 1;
    RETAINTEST_RETAIN_ARRAYSIMPLESTRUCTURE[3].SIMPLE_REAL := RETAINTEST_RETAIN_ARRAYSIMPLESTRUCTURE[3].SIMPLE_REAL + 1.1;
    RETAINTEST_RETAIN_ARRAYSIMPLESTRUCTURE[3].SIMPLE_SINT := RETAINTEST_RETAIN_ARRAYSIMPLESTRUCTURE[3].SIMPLE_SINT + 1;
    RETAINTEST_RETAIN_ARRAYSIMPLESTRUCTURE[3].SIMPLE_STRING := ANY_TO_STRING(RETAINTEST_RETAIN_ARRAYSIMPLESTRUCTURE[3].SIMPLE_DINT) + ' ' + ANY_TO_STRING(RETAINTEST_RETAIN_ARRAYSIMPLESTRUCTURE[3].SIMPLE_TIME);
    RETAINTEST_RETAIN_ARRAYSIMPLESTRUCTURE[3].SIMPLE_TIME := RETAINTEST_RETAIN_ARRAYSIMPLESTRUCTURE[3].SIMPLE_TIME + PULSE_TIME;
    RETAINTEST_RETAIN_ARRAYSIMPLESTRUCTURE[3].SIMPLE_UDINT := RETAINTEST_RETAIN_ARRAYSIMPLESTRUCTURE[3].SIMPLE_UDINT + 1;
    RETAINTEST_RETAIN_ARRAYSIMPLESTRUCTURE[3].SIMPLE_UINT := RETAINTEST_RETAIN_ARRAYSIMPLESTRUCTURE[3].SIMPLE_UINT + 1;
    RETAINTEST_RETAIN_ARRAYSIMPLESTRUCTURE[3].SIMPLE_ULINT := RETAINTEST_RETAIN_ARRAYSIMPLESTRUCTURE[3].SIMPLE_ULINT + 1;
    RETAINTEST_RETAIN_ARRAYSIMPLESTRUCTURE[3].SIMPLE_USINT := RETAINTEST_RETAIN_ARRAYSIMPLESTRUCTURE[3].SIMPLE_USINT + 1;
    RETAINTEST_RETAIN_ARRAYSIMPLESTRUCTURE[3].SIMPLE_WORD := RETAINTEST_RETAIN_ARRAYSIMPLESTRUCTURE[3].SIMPLE_WORD + 1;

    RETAINTEST_RETAIN_ARRAYSIMPLESTRUCTURE[4].SIMPLE_BOOL := NOT RETAINTEST_RETAIN_ARRAYSIMPLESTRUCTURE[4].SIMPLE_BOOL;
    RETAINTEST_RETAIN_ARRAYSIMPLESTRUCTURE[4].SIMPLE_BYTE := RETAINTEST_RETAIN_ARRAYSIMPLESTRUCTURE[4].SIMPLE_BYTE + 1;
    RETAINTEST_RETAIN_ARRAYSIMPLESTRUCTURE[4].SIMPLE_DATE := ANY_TO_DATE(1445385600 + RETAINTEST_RETAIN_ARRAYSIMPLESTRUCTURE[4].SIMPLE_DINT * 86400);
    RETAINTEST_RETAIN_ARRAYSIMPLESTRUCTURE[4].SIMPLE_DINT := RETAINTEST_RETAIN_ARRAYSIMPLESTRUCTURE[4].SIMPLE_DINT + 1;
    RETAINTEST_RETAIN_ARRAYSIMPLESTRUCTURE[4].SIMPLE_DWORD := RETAINTEST_RETAIN_ARRAYSIMPLESTRUCTURE[4].SIMPLE_DWORD + 1;
    RETAINTEST_RETAIN_ARRAYSIMPLESTRUCTURE[4].SIMPLE_INT := RETAINTEST_RETAIN_ARRAYSIMPLESTRUCTURE[4].SIMPLE_INT + 1;
    RETAINTEST_RETAIN_ARRAYSIMPLESTRUCTURE[4].SIMPLE_LINT := RETAINTEST_RETAIN_ARRAYSIMPLESTRUCTURE[4].SIMPLE_LINT + 1;
    RETAINTEST_RETAIN_ARRAYSIMPLESTRUCTURE[4].SIMPLE_LREAL := RETAINTEST_RETAIN_ARRAYSIMPLESTRUCTURE[4].SIMPLE_LREAL + 1.1;
    RETAINTEST_RETAIN_ARRAYSIMPLESTRUCTURE[4].SIMPLE_LWORD := RETAINTEST_RETAIN_ARRAYSIMPLESTRUCTURE[4].SIMPLE_LWORD + 1;
    RETAINTEST_RETAIN_ARRAYSIMPLESTRUCTURE[4].SIMPLE_REAL := RETAINTEST_RETAIN_ARRAYSIMPLESTRUCTURE[4].SIMPLE_REAL + 1.1;
    RETAINTEST_RETAIN_ARRAYSIMPLESTRUCTURE[4].SIMPLE_SINT := RETAINTEST_RETAIN_ARRAYSIMPLESTRUCTURE[4].SIMPLE_SINT + 1;
    RETAINTEST_RETAIN_ARRAYSIMPLESTRUCTURE[4].SIMPLE_STRING := ANY_TO_STRING(RETAINTEST_RETAIN_ARRAYSIMPLESTRUCTURE[4].SIMPLE_DINT) + ' ' + ANY_TO_STRING(RETAINTEST_RETAIN_ARRAYSIMPLESTRUCTURE[4].SIMPLE_TIME);
    RETAINTEST_RETAIN_ARRAYSIMPLESTRUCTURE[4].SIMPLE_TIME := RETAINTEST_RETAIN_ARRAYSIMPLESTRUCTURE[4].SIMPLE_TIME + PULSE_TIME;
    RETAINTEST_RETAIN_ARRAYSIMPLESTRUCTURE[4].SIMPLE_UDINT := RETAINTEST_RETAIN_ARRAYSIMPLESTRUCTURE[4].SIMPLE_UDINT + 1;
    RETAINTEST_RETAIN_ARRAYSIMPLESTRUCTURE[4].SIMPLE_UINT := RETAINTEST_RETAIN_ARRAYSIMPLESTRUCTURE[4].SIMPLE_UINT + 1;
    RETAINTEST_RETAIN_ARRAYSIMPLESTRUCTURE[4].SIMPLE_ULINT := RETAINTEST_RETAIN_ARRAYSIMPLESTRUCTURE[4].SIMPLE_ULINT + 1;
    RETAINTEST_RETAIN_ARRAYSIMPLESTRUCTURE[4].SIMPLE_USINT := RETAINTEST_RETAIN_ARRAYSIMPLESTRUCTURE[4].SIMPLE_USINT + 1;
    RETAINTEST_RETAIN_ARRAYSIMPLESTRUCTURE[4].SIMPLE_WORD := RETAINTEST_RETAIN_ARRAYSIMPLESTRUCTURE[4].SIMPLE_WORD + 1;

    RETAINTEST_RETAIN_ARRAYSIMPLESTRUCTURE[5].SIMPLE_BOOL := RETAINTEST_RETAIN_ARRAYSIMPLESTRUCTURE[4].SIMPLE_BOOL;
    RETAINTEST_RETAIN_ARRAYSIMPLESTRUCTURE[5].SIMPLE_BYTE := RETAINTEST_RETAIN_ARRAYSIMPLESTRUCTURE[4].SIMPLE_BYTE;
    RETAINTEST_RETAIN_ARRAYSIMPLESTRUCTURE[5].SIMPLE_DATE := RETAINTEST_RETAIN_ARRAYSIMPLESTRUCTURE[4].SIMPLE_DATE;
    RETAINTEST_RETAIN_ARRAYSIMPLESTRUCTURE[5].SIMPLE_DINT := RETAINTEST_RETAIN_ARRAYSIMPLESTRUCTURE[4].SIMPLE_DINT;
    RETAINTEST_RETAIN_ARRAYSIMPLESTRUCTURE[5].SIMPLE_DWORD := RETAINTEST_RETAIN_ARRAYSIMPLESTRUCTURE[4].SIMPLE_DWORD;
    RETAINTEST_RETAIN_ARRAYSIMPLESTRUCTURE[5].SIMPLE_INT := RETAINTEST_RETAIN_ARRAYSIMPLESTRUCTURE[4].SIMPLE_INT;
    RETAINTEST_RETAIN_ARRAYSIMPLESTRUCTURE[5].SIMPLE_LINT := RETAINTEST_RETAIN_ARRAYSIMPLESTRUCTURE[4].SIMPLE_LINT;
    RETAINTEST_RETAIN_ARRAYSIMPLESTRUCTURE[5].SIMPLE_LREAL := RETAINTEST_RETAIN_ARRAYSIMPLESTRUCTURE[4].SIMPLE_LREAL;
    RETAINTEST_RETAIN_ARRAYSIMPLESTRUCTURE[5].SIMPLE_LWORD := RETAINTEST_RETAIN_ARRAYSIMPLESTRUCTURE[4].SIMPLE_LWORD;
    RETAINTEST_RETAIN_ARRAYSIMPLESTRUCTURE[5].SIMPLE_REAL := RETAINTEST_RETAIN_ARRAYSIMPLESTRUCTURE[4].SIMPLE_REAL;
    RETAINTEST_RETAIN_ARRAYSIMPLESTRUCTURE[5].SIMPLE_SINT := RETAINTEST_RETAIN_ARRAYSIMPLESTRUCTURE[4].SIMPLE_SINT;
    RETAINTEST_RETAIN_ARRAYSIMPLESTRUCTURE[5].SIMPLE_STRING := RETAINTEST_RETAIN_ARRAYSIMPLESTRUCTURE[4].SIMPLE_STRING;
    RETAINTEST_RETAIN_ARRAYSIMPLESTRUCTURE[5].SIMPLE_TIME := RETAINTEST_RETAIN_ARRAYSIMPLESTRUCTURE[4].SIMPLE_TIME;
    RETAINTEST_RETAIN_ARRAYSIMPLESTRUCTURE[5].SIMPLE_UDINT := RETAINTEST_RETAIN_ARRAYSIMPLESTRUCTURE[4].SIMPLE_UDINT;
    RETAINTEST_RETAIN_ARRAYSIMPLESTRUCTURE[5].SIMPLE_UINT := RETAINTEST_RETAIN_ARRAYSIMPLESTRUCTURE[4].SIMPLE_UINT;
    RETAINTEST_RETAIN_ARRAYSIMPLESTRUCTURE[5].SIMPLE_ULINT := RETAINTEST_RETAIN_ARRAYSIMPLESTRUCTURE[4].SIMPLE_ULINT;
    RETAINTEST_RETAIN_ARRAYSIMPLESTRUCTURE[5].SIMPLE_USINT := RETAINTEST_RETAIN_ARRAYSIMPLESTRUCTURE[4].SIMPLE_USINT;
    RETAINTEST_RETAIN_ARRAYSIMPLESTRUCTURE[5].SIMPLE_WORD := RETAINTEST_RETAIN_ARRAYSIMPLESTRUCTURE[4].SIMPLE_WORD;

    RETAINTEST_NONRETAIN_ARRAYSIMPLESTRUCTURE[0].SIMPLE_BOOL := NOT RETAINTEST_NONRETAIN_ARRAYSIMPLESTRUCTURE[0].SIMPLE_BOOL;
    RETAINTEST_NONRETAIN_ARRAYSIMPLESTRUCTURE[0].SIMPLE_BYTE := RETAINTEST_NONRETAIN_ARRAYSIMPLESTRUCTURE[0].SIMPLE_BYTE + 1;
    RETAINTEST_NONRETAIN_ARRAYSIMPLESTRUCTURE[0].SIMPLE_DATE := ANY_TO_DATE(1445385600 + RETAINTEST_NONRETAIN_ARRAYSIMPLESTRUCTURE[0].SIMPLE_DINT * 86400);
    RETAINTEST_NONRETAIN_ARRAYSIMPLESTRUCTURE[0].SIMPLE_DINT := RETAINTEST_NONRETAIN_ARRAYSIMPLESTRUCTURE[0].SIMPLE_DINT + 1;
    RETAINTEST_NONRETAIN_ARRAYSIMPLESTRUCTURE[0].SIMPLE_DWORD := RETAINTEST_NONRETAIN_ARRAYSIMPLESTRUCTURE[0].SIMPLE_DWORD + 1;
    RETAINTEST_NONRETAIN_ARRAYSIMPLESTRUCTURE[0].SIMPLE_INT := RETAINTEST_NONRETAIN_ARRAYSIMPLESTRUCTURE[0].SIMPLE_INT + 1;
    RETAINTEST_NONRETAIN_ARRAYSIMPLESTRUCTURE[0].SIMPLE_LINT := RETAINTEST_NONRETAIN_ARRAYSIMPLESTRUCTURE[0].SIMPLE_LINT + 1;
    RETAINTEST_NONRETAIN_ARRAYSIMPLESTRUCTURE[0].SIMPLE_LREAL := RETAINTEST_NONRETAIN_ARRAYSIMPLESTRUCTURE[0].SIMPLE_LREAL + 1.1;
    RETAINTEST_NONRETAIN_ARRAYSIMPLESTRUCTURE[0].SIMPLE_LWORD := RETAINTEST_NONRETAIN_ARRAYSIMPLESTRUCTURE[0].SIMPLE_LWORD + 1;
    RETAINTEST_NONRETAIN_ARRAYSIMPLESTRUCTURE[0].SIMPLE_REAL := RETAINTEST_NONRETAIN_ARRAYSIMPLESTRUCTURE[0].SIMPLE_REAL + 1.1;
    RETAINTEST_NONRETAIN_ARRAYSIMPLESTRUCTURE[0].SIMPLE_SINT := RETAINTEST_NONRETAIN_ARRAYSIMPLESTRUCTURE[0].SIMPLE_SINT + 1;
    RETAINTEST_NONRETAIN_ARRAYSIMPLESTRUCTURE[0].SIMPLE_STRING := ANY_TO_STRING(RETAINTEST_NONRETAIN_ARRAYSIMPLESTRUCTURE[0].SIMPLE_DINT) + ' ' + ANY_TO_STRING(RETAINTEST_NONRETAIN_ARRAYSIMPLESTRUCTURE[0].SIMPLE_TIME);
    RETAINTEST_NONRETAIN_ARRAYSIMPLESTRUCTURE[0].SIMPLE_TIME := RETAINTEST_NONRETAIN_ARRAYSIMPLESTRUCTURE[0].SIMPLE_TIME + PULSE_TIME;
    RETAINTEST_NONRETAIN_ARRAYSIMPLESTRUCTURE[0].SIMPLE_UDINT := RETAINTEST_NONRETAIN_ARRAYSIMPLESTRUCTURE[0].SIMPLE_UDINT + 1;
    RETAINTEST_NONRETAIN_ARRAYSIMPLESTRUCTURE[0].SIMPLE_UINT := RETAINTEST_NONRETAIN_ARRAYSIMPLESTRUCTURE[0].SIMPLE_UINT + 1;
    RETAINTEST_NONRETAIN_ARRAYSIMPLESTRUCTURE[0].SIMPLE_ULINT := RETAINTEST_NONRETAIN_ARRAYSIMPLESTRUCTURE[0].SIMPLE_ULINT + 1;
    RETAINTEST_NONRETAIN_ARRAYSIMPLESTRUCTURE[0].SIMPLE_USINT := RETAINTEST_NONRETAIN_ARRAYSIMPLESTRUCTURE[0].SIMPLE_USINT + 1;
    RETAINTEST_NONRETAIN_ARRAYSIMPLESTRUCTURE[0].SIMPLE_WORD := RETAINTEST_NONRETAIN_ARRAYSIMPLESTRUCTURE[0].SIMPLE_WORD + 1;

    RETAINTEST_NONRETAIN_ARRAYSIMPLESTRUCTURE[1].SIMPLE_BOOL := NOT RETAINTEST_NONRETAIN_ARRAYSIMPLESTRUCTURE[1].SIMPLE_BOOL;
    RETAINTEST_NONRETAIN_ARRAYSIMPLESTRUCTURE[1].SIMPLE_BYTE := RETAINTEST_NONRETAIN_ARRAYSIMPLESTRUCTURE[1].SIMPLE_BYTE + 1;
    RETAINTEST_NONRETAIN_ARRAYSIMPLESTRUCTURE[1].SIMPLE_DATE := ANY_TO_DATE(1445385600 + RETAINTEST_NONRETAIN_ARRAYSIMPLESTRUCTURE[1].SIMPLE_DINT * 86400);
    RETAINTEST_NONRETAIN_ARRAYSIMPLESTRUCTURE[1].SIMPLE_DINT := RETAINTEST_NONRETAIN_ARRAYSIMPLESTRUCTURE[1].SIMPLE_DINT + 1;
    RETAINTEST_NONRETAIN_ARRAYSIMPLESTRUCTURE[1].SIMPLE_DWORD := RETAINTEST_NONRETAIN_ARRAYSIMPLESTRUCTURE[1].SIMPLE_DWORD + 1;
    RETAINTEST_NONRETAIN_ARRAYSIMPLESTRUCTURE[1].SIMPLE_INT := RETAINTEST_NONRETAIN_ARRAYSIMPLESTRUCTURE[1].SIMPLE_INT + 1;
    RETAINTEST_NONRETAIN_ARRAYSIMPLESTRUCTURE[1].SIMPLE_LINT := RETAINTEST_NONRETAIN_ARRAYSIMPLESTRUCTURE[1].SIMPLE_LINT + 1;
    RETAINTEST_NONRETAIN_ARRAYSIMPLESTRUCTURE[1].SIMPLE_LREAL := RETAINTEST_NONRETAIN_ARRAYSIMPLESTRUCTURE[1].SIMPLE_LREAL + 1.1;
    RETAINTEST_NONRETAIN_ARRAYSIMPLESTRUCTURE[1].SIMPLE_LWORD := RETAINTEST_NONRETAIN_ARRAYSIMPLESTRUCTURE[1].SIMPLE_LWORD + 1;
    RETAINTEST_NONRETAIN_ARRAYSIMPLESTRUCTURE[1].SIMPLE_REAL := RETAINTEST_NONRETAIN_ARRAYSIMPLESTRUCTURE[1].SIMPLE_REAL + 1.1;
    RETAINTEST_NONRETAIN_ARRAYSIMPLESTRUCTURE[1].SIMPLE_SINT := RETAINTEST_NONRETAIN_ARRAYSIMPLESTRUCTURE[1].SIMPLE_SINT + 1;
    RETAINTEST_NONRETAIN_ARRAYSIMPLESTRUCTURE[1].SIMPLE_STRING := ANY_TO_STRING(RETAINTEST_NONRETAIN_ARRAYSIMPLESTRUCTURE[1].SIMPLE_DINT) + ' ' + ANY_TO_STRING(RETAINTEST_NONRETAIN_ARRAYSIMPLESTRUCTURE[1].SIMPLE_TIME);
    RETAINTEST_NONRETAIN_ARRAYSIMPLESTRUCTURE[1].SIMPLE_TIME := RETAINTEST_NONRETAIN_ARRAYSIMPLESTRUCTURE[1].SIMPLE_TIME + PULSE_TIME;
    RETAINTEST_NONRETAIN_ARRAYSIMPLESTRUCTURE[1].SIMPLE_UDINT := RETAINTEST_NONRETAIN_ARRAYSIMPLESTRUCTURE[1].SIMPLE_UDINT + 1;
    RETAINTEST_NONRETAIN_ARRAYSIMPLESTRUCTURE[1].SIMPLE_UINT := RETAINTEST_NONRETAIN_ARRAYSIMPLESTRUCTURE[1].SIMPLE_UINT + 1;
    RETAINTEST_NONRETAIN_ARRAYSIMPLESTRUCTURE[1].SIMPLE_ULINT := RETAINTEST_NONRETAIN_ARRAYSIMPLESTRUCTURE[1].SIMPLE_ULINT + 1;
    RETAINTEST_NONRETAIN_ARRAYSIMPLESTRUCTURE[1].SIMPLE_USINT := RETAINTEST_NONRETAIN_ARRAYSIMPLESTRUCTURE[1].SIMPLE_USINT + 1;
    RETAINTEST_NONRETAIN_ARRAYSIMPLESTRUCTURE[1].SIMPLE_WORD := RETAINTEST_NONRETAIN_ARRAYSIMPLESTRUCTURE[1].SIMPLE_WORD + 1;

    RETAINTEST_NONRETAIN_ARRAYSIMPLESTRUCTURE[2].SIMPLE_BOOL := NOT RETAINTEST_NONRETAIN_ARRAYSIMPLESTRUCTURE[2].SIMPLE_BOOL;
    RETAINTEST_NONRETAIN_ARRAYSIMPLESTRUCTURE[2].SIMPLE_BYTE := RETAINTEST_NONRETAIN_ARRAYSIMPLESTRUCTURE[2].SIMPLE_BYTE + 1;
    RETAINTEST_NONRETAIN_ARRAYSIMPLESTRUCTURE[2].SIMPLE_DATE := ANY_TO_DATE(1445385600 + RETAINTEST_NONRETAIN_ARRAYSIMPLESTRUCTURE[2].SIMPLE_DINT * 86400);
    RETAINTEST_NONRETAIN_ARRAYSIMPLESTRUCTURE[2].SIMPLE_DINT := RETAINTEST_NONRETAIN_ARRAYSIMPLESTRUCTURE[2].SIMPLE_DINT + 1;
    RETAINTEST_NONRETAIN_ARRAYSIMPLESTRUCTURE[2].SIMPLE_DWORD := RETAINTEST_NONRETAIN_ARRAYSIMPLESTRUCTURE[2].SIMPLE_DWORD + 1;
    RETAINTEST_NONRETAIN_ARRAYSIMPLESTRUCTURE[2].SIMPLE_INT := RETAINTEST_NONRETAIN_ARRAYSIMPLESTRUCTURE[2].SIMPLE_INT + 1;
    RETAINTEST_NONRETAIN_ARRAYSIMPLESTRUCTURE[2].SIMPLE_LINT := RETAINTEST_NONRETAIN_ARRAYSIMPLESTRUCTURE[2].SIMPLE_LINT + 1;
    RETAINTEST_NONRETAIN_ARRAYSIMPLESTRUCTURE[2].SIMPLE_LREAL := RETAINTEST_NONRETAIN_ARRAYSIMPLESTRUCTURE[2].SIMPLE_LREAL + 1.1;
    RETAINTEST_NONRETAIN_ARRAYSIMPLESTRUCTURE[2].SIMPLE_LWORD := RETAINTEST_NONRETAIN_ARRAYSIMPLESTRUCTURE[2].SIMPLE_LWORD + 1;
    RETAINTEST_NONRETAIN_ARRAYSIMPLESTRUCTURE[2].SIMPLE_REAL := RETAINTEST_NONRETAIN_ARRAYSIMPLESTRUCTURE[2].SIMPLE_REAL + 1.1;
    RETAINTEST_NONRETAIN_ARRAYSIMPLESTRUCTURE[2].SIMPLE_SINT := RETAINTEST_NONRETAIN_ARRAYSIMPLESTRUCTURE[2].SIMPLE_SINT + 1;
    RETAINTEST_NONRETAIN_ARRAYSIMPLESTRUCTURE[2].SIMPLE_STRING := ANY_TO_STRING(RETAINTEST_NONRETAIN_ARRAYSIMPLESTRUCTURE[2].SIMPLE_DINT) + ' ' + ANY_TO_STRING(RETAINTEST_NONRETAIN_ARRAYSIMPLESTRUCTURE[2].SIMPLE_TIME);
    RETAINTEST_NONRETAIN_ARRAYSIMPLESTRUCTURE[2].SIMPLE_TIME := RETAINTEST_NONRETAIN_ARRAYSIMPLESTRUCTURE[2].SIMPLE_TIME + PULSE_TIME;
    RETAINTEST_NONRETAIN_ARRAYSIMPLESTRUCTURE[2].SIMPLE_UDINT := RETAINTEST_NONRETAIN_ARRAYSIMPLESTRUCTURE[2].SIMPLE_UDINT + 1;
    RETAINTEST_NONRETAIN_ARRAYSIMPLESTRUCTURE[2].SIMPLE_UINT := RETAINTEST_NONRETAIN_ARRAYSIMPLESTRUCTURE[2].SIMPLE_UINT + 1;
    RETAINTEST_NONRETAIN_ARRAYSIMPLESTRUCTURE[2].SIMPLE_ULINT := RETAINTEST_NONRETAIN_ARRAYSIMPLESTRUCTURE[2].SIMPLE_ULINT + 1;
    RETAINTEST_NONRETAIN_ARRAYSIMPLESTRUCTURE[2].SIMPLE_USINT := RETAINTEST_NONRETAIN_ARRAYSIMPLESTRUCTURE[2].SIMPLE_USINT + 1;
    RETAINTEST_NONRETAIN_ARRAYSIMPLESTRUCTURE[2].SIMPLE_WORD := RETAINTEST_NONRETAIN_ARRAYSIMPLESTRUCTURE[2].SIMPLE_WORD + 1;

    RETAINTEST_NONRETAIN_ARRAYSIMPLESTRUCTURE[3].SIMPLE_BOOL := NOT RETAINTEST_NONRETAIN_ARRAYSIMPLESTRUCTURE[3].SIMPLE_BOOL;
    RETAINTEST_NONRETAIN_ARRAYSIMPLESTRUCTURE[3].SIMPLE_BYTE := RETAINTEST_NONRETAIN_ARRAYSIMPLESTRUCTURE[3].SIMPLE_BYTE + 1;
    RETAINTEST_NONRETAIN_ARRAYSIMPLESTRUCTURE[3].SIMPLE_DATE := ANY_TO_DATE(1445385600 + RETAINTEST_NONRETAIN_ARRAYSIMPLESTRUCTURE[3].SIMPLE_DINT * 86400);
    RETAINTEST_NONRETAIN_ARRAYSIMPLESTRUCTURE[3].SIMPLE_DINT := RETAINTEST_NONRETAIN_ARRAYSIMPLESTRUCTURE[3].SIMPLE_DINT + 1;
    RETAINTEST_NONRETAIN_ARRAYSIMPLESTRUCTURE[3].SIMPLE_DWORD := RETAINTEST_NONRETAIN_ARRAYSIMPLESTRUCTURE[3].SIMPLE_DWORD + 1;
    RETAINTEST_NONRETAIN_ARRAYSIMPLESTRUCTURE[3].SIMPLE_INT := RETAINTEST_NONRETAIN_ARRAYSIMPLESTRUCTURE[3].SIMPLE_INT + 1;
    RETAINTEST_NONRETAIN_ARRAYSIMPLESTRUCTURE[3].SIMPLE_LINT := RETAINTEST_NONRETAIN_ARRAYSIMPLESTRUCTURE[3].SIMPLE_LINT + 1;
    RETAINTEST_NONRETAIN_ARRAYSIMPLESTRUCTURE[3].SIMPLE_LREAL := RETAINTEST_NONRETAIN_ARRAYSIMPLESTRUCTURE[3].SIMPLE_LREAL + 1.1;
    RETAINTEST_NONRETAIN_ARRAYSIMPLESTRUCTURE[3].SIMPLE_LWORD := RETAINTEST_NONRETAIN_ARRAYSIMPLESTRUCTURE[3].SIMPLE_LWORD + 1;
    RETAINTEST_NONRETAIN_ARRAYSIMPLESTRUCTURE[3].SIMPLE_REAL := RETAINTEST_NONRETAIN_ARRAYSIMPLESTRUCTURE[3].SIMPLE_REAL + 1.1;
    RETAINTEST_NONRETAIN_ARRAYSIMPLESTRUCTURE[3].SIMPLE_SINT := RETAINTEST_NONRETAIN_ARRAYSIMPLESTRUCTURE[3].SIMPLE_SINT + 1;
    RETAINTEST_NONRETAIN_ARRAYSIMPLESTRUCTURE[3].SIMPLE_STRING := ANY_TO_STRING(RETAINTEST_NONRETAIN_ARRAYSIMPLESTRUCTURE[3].SIMPLE_DINT) + ' ' + ANY_TO_STRING(RETAINTEST_NONRETAIN_ARRAYSIMPLESTRUCTURE[3].SIMPLE_TIME);
    RETAINTEST_NONRETAIN_ARRAYSIMPLESTRUCTURE[3].SIMPLE_TIME := RETAINTEST_NONRETAIN_ARRAYSIMPLESTRUCTURE[3].SIMPLE_TIME + PULSE_TIME;
    RETAINTEST_NONRETAIN_ARRAYSIMPLESTRUCTURE[3].SIMPLE_UDINT := RETAINTEST_NONRETAIN_ARRAYSIMPLESTRUCTURE[3].SIMPLE_UDINT + 1;
    RETAINTEST_NONRETAIN_ARRAYSIMPLESTRUCTURE[3].SIMPLE_UINT := RETAINTEST_NONRETAIN_ARRAYSIMPLESTRUCTURE[3].SIMPLE_UINT + 1;
    RETAINTEST_NONRETAIN_ARRAYSIMPLESTRUCTURE[3].SIMPLE_ULINT := RETAINTEST_NONRETAIN_ARRAYSIMPLESTRUCTURE[3].SIMPLE_ULINT + 1;
    RETAINTEST_NONRETAIN_ARRAYSIMPLESTRUCTURE[3].SIMPLE_USINT := RETAINTEST_NONRETAIN_ARRAYSIMPLESTRUCTURE[3].SIMPLE_USINT + 1;
    RETAINTEST_NONRETAIN_ARRAYSIMPLESTRUCTURE[3].SIMPLE_WORD := RETAINTEST_NONRETAIN_ARRAYSIMPLESTRUCTURE[3].SIMPLE_WORD + 1;

    RETAINTEST_NONRETAIN_ARRAYSIMPLESTRUCTURE[4].SIMPLE_BOOL := NOT RETAINTEST_NONRETAIN_ARRAYSIMPLESTRUCTURE[4].SIMPLE_BOOL;
    RETAINTEST_NONRETAIN_ARRAYSIMPLESTRUCTURE[4].SIMPLE_BYTE := RETAINTEST_NONRETAIN_ARRAYSIMPLESTRUCTURE[4].SIMPLE_BYTE + 1;
    RETAINTEST_NONRETAIN_ARRAYSIMPLESTRUCTURE[4].SIMPLE_DATE := ANY_TO_DATE(1445385600 + RETAINTEST_NONRETAIN_ARRAYSIMPLESTRUCTURE[4].SIMPLE_DINT * 86400);
    RETAINTEST_NONRETAIN_ARRAYSIMPLESTRUCTURE[4].SIMPLE_DINT := RETAINTEST_NONRETAIN_ARRAYSIMPLESTRUCTURE[4].SIMPLE_DINT + 1;
    RETAINTEST_NONRETAIN_ARRAYSIMPLESTRUCTURE[4].SIMPLE_DWORD := RETAINTEST_NONRETAIN_ARRAYSIMPLESTRUCTURE[4].SIMPLE_DWORD + 1;
    RETAINTEST_NONRETAIN_ARRAYSIMPLESTRUCTURE[4].SIMPLE_INT := RETAINTEST_NONRETAIN_ARRAYSIMPLESTRUCTURE[4].SIMPLE_INT + 1;
    RETAINTEST_NONRETAIN_ARRAYSIMPLESTRUCTURE[4].SIMPLE_LINT := RETAINTEST_NONRETAIN_ARRAYSIMPLESTRUCTURE[4].SIMPLE_LINT + 1;
    RETAINTEST_NONRETAIN_ARRAYSIMPLESTRUCTURE[4].SIMPLE_LREAL := RETAINTEST_NONRETAIN_ARRAYSIMPLESTRUCTURE[4].SIMPLE_LREAL + 1.1;
    RETAINTEST_NONRETAIN_ARRAYSIMPLESTRUCTURE[4].SIMPLE_LWORD := RETAINTEST_NONRETAIN_ARRAYSIMPLESTRUCTURE[4].SIMPLE_LWORD + 1;
    RETAINTEST_NONRETAIN_ARRAYSIMPLESTRUCTURE[4].SIMPLE_REAL := RETAINTEST_NONRETAIN_ARRAYSIMPLESTRUCTURE[4].SIMPLE_REAL + 1.1;
    RETAINTEST_NONRETAIN_ARRAYSIMPLESTRUCTURE[4].SIMPLE_SINT := RETAINTEST_NONRETAIN_ARRAYSIMPLESTRUCTURE[4].SIMPLE_SINT + 1;
    RETAINTEST_NONRETAIN_ARRAYSIMPLESTRUCTURE[4].SIMPLE_STRING := ANY_TO_STRING(RETAINTEST_NONRETAIN_ARRAYSIMPLESTRUCTURE[4].SIMPLE_DINT) + ' ' + ANY_TO_STRING(RETAINTEST_NONRETAIN_ARRAYSIMPLESTRUCTURE[4].SIMPLE_TIME);
    RETAINTEST_NONRETAIN_ARRAYSIMPLESTRUCTURE[4].SIMPLE_TIME := RETAINTEST_NONRETAIN_ARRAYSIMPLESTRUCTURE[4].SIMPLE_TIME + PULSE_TIME;
    RETAINTEST_NONRETAIN_ARRAYSIMPLESTRUCTURE[4].SIMPLE_UDINT := RETAINTEST_NONRETAIN_ARRAYSIMPLESTRUCTURE[4].SIMPLE_UDINT + 1;
    RETAINTEST_NONRETAIN_ARRAYSIMPLESTRUCTURE[4].SIMPLE_UINT := RETAINTEST_NONRETAIN_ARRAYSIMPLESTRUCTURE[4].SIMPLE_UINT + 1;
    RETAINTEST_NONRETAIN_ARRAYSIMPLESTRUCTURE[4].SIMPLE_ULINT := RETAINTEST_NONRETAIN_ARRAYSIMPLESTRUCTURE[4].SIMPLE_ULINT + 1;
    RETAINTEST_NONRETAIN_ARRAYSIMPLESTRUCTURE[4].SIMPLE_USINT := RETAINTEST_NONRETAIN_ARRAYSIMPLESTRUCTURE[4].SIMPLE_USINT + 1;
    RETAINTEST_NONRETAIN_ARRAYSIMPLESTRUCTURE[4].SIMPLE_WORD := RETAINTEST_NONRETAIN_ARRAYSIMPLESTRUCTURE[4].SIMPLE_WORD + 1;

    RETAINTEST_NONRETAIN_ARRAYSIMPLESTRUCTURE[5].SIMPLE_BOOL := RETAINTEST_NONRETAIN_ARRAYSIMPLESTRUCTURE[4].SIMPLE_BOOL;
    RETAINTEST_NONRETAIN_ARRAYSIMPLESTRUCTURE[5].SIMPLE_BYTE := RETAINTEST_NONRETAIN_ARRAYSIMPLESTRUCTURE[4].SIMPLE_BYTE;
    RETAINTEST_NONRETAIN_ARRAYSIMPLESTRUCTURE[5].SIMPLE_DATE := RETAINTEST_NONRETAIN_ARRAYSIMPLESTRUCTURE[4].SIMPLE_DATE;
    RETAINTEST_NONRETAIN_ARRAYSIMPLESTRUCTURE[5].SIMPLE_DINT := RETAINTEST_NONRETAIN_ARRAYSIMPLESTRUCTURE[4].SIMPLE_DINT;
    RETAINTEST_NONRETAIN_ARRAYSIMPLESTRUCTURE[5].SIMPLE_DWORD := RETAINTEST_NONRETAIN_ARRAYSIMPLESTRUCTURE[4].SIMPLE_DWORD;
    RETAINTEST_NONRETAIN_ARRAYSIMPLESTRUCTURE[5].SIMPLE_INT := RETAINTEST_NONRETAIN_ARRAYSIMPLESTRUCTURE[4].SIMPLE_INT;
    RETAINTEST_NONRETAIN_ARRAYSIMPLESTRUCTURE[5].SIMPLE_LINT := RETAINTEST_NONRETAIN_ARRAYSIMPLESTRUCTURE[4].SIMPLE_LINT;
    RETAINTEST_NONRETAIN_ARRAYSIMPLESTRUCTURE[5].SIMPLE_LREAL := RETAINTEST_NONRETAIN_ARRAYSIMPLESTRUCTURE[4].SIMPLE_LREAL;
    RETAINTEST_NONRETAIN_ARRAYSIMPLESTRUCTURE[5].SIMPLE_LWORD := RETAINTEST_NONRETAIN_ARRAYSIMPLESTRUCTURE[4].SIMPLE_LWORD;
    RETAINTEST_NONRETAIN_ARRAYSIMPLESTRUCTURE[5].SIMPLE_REAL := RETAINTEST_NONRETAIN_ARRAYSIMPLESTRUCTURE[4].SIMPLE_REAL;
    RETAINTEST_NONRETAIN_ARRAYSIMPLESTRUCTURE[5].SIMPLE_SINT := RETAINTEST_NONRETAIN_ARRAYSIMPLESTRUCTURE[4].SIMPLE_SINT;
    RETAINTEST_NONRETAIN_ARRAYSIMPLESTRUCTURE[5].SIMPLE_STRING := RETAINTEST_NONRETAIN_ARRAYSIMPLESTRUCTURE[4].SIMPLE_STRING;
    RETAINTEST_NONRETAIN_ARRAYSIMPLESTRUCTURE[5].SIMPLE_TIME := RETAINTEST_NONRETAIN_ARRAYSIMPLESTRUCTURE[4].SIMPLE_TIME;
    RETAINTEST_NONRETAIN_ARRAYSIMPLESTRUCTURE[5].SIMPLE_UDINT := RETAINTEST_NONRETAIN_ARRAYSIMPLESTRUCTURE[4].SIMPLE_UDINT;
    RETAINTEST_NONRETAIN_ARRAYSIMPLESTRUCTURE[5].SIMPLE_UINT := RETAINTEST_NONRETAIN_ARRAYSIMPLESTRUCTURE[4].SIMPLE_UINT;
    RETAINTEST_NONRETAIN_ARRAYSIMPLESTRUCTURE[5].SIMPLE_ULINT := RETAINTEST_NONRETAIN_ARRAYSIMPLESTRUCTURE[4].SIMPLE_ULINT;
    RETAINTEST_NONRETAIN_ARRAYSIMPLESTRUCTURE[5].SIMPLE_USINT := RETAINTEST_NONRETAIN_ARRAYSIMPLESTRUCTURE[4].SIMPLE_USINT;
    RETAINTEST_NONRETAIN_ARRAYSIMPLESTRUCTURE[5].SIMPLE_WORD := RETAINTEST_NONRETAIN_ARRAYSIMPLESTRUCTURE[4].SIMPLE_WORD;

    RETAINTEST_AUTO_ARRAYSIMPLESTRUCTURE[0].SIMPLE_BOOL := NOT RETAINTEST_AUTO_ARRAYSIMPLESTRUCTURE[0].SIMPLE_BOOL;
    RETAINTEST_AUTO_ARRAYSIMPLESTRUCTURE[0].SIMPLE_BYTE := RETAINTEST_AUTO_ARRAYSIMPLESTRUCTURE[0].SIMPLE_BYTE + 1;
    RETAINTEST_AUTO_ARRAYSIMPLESTRUCTURE[0].SIMPLE_DATE := ANY_TO_DATE(1445385600 + RETAINTEST_AUTO_ARRAYSIMPLESTRUCTURE[0].SIMPLE_DINT * 86400);
    RETAINTEST_AUTO_ARRAYSIMPLESTRUCTURE[0].SIMPLE_DINT := RETAINTEST_AUTO_ARRAYSIMPLESTRUCTURE[0].SIMPLE_DINT + 1;
    RETAINTEST_AUTO_ARRAYSIMPLESTRUCTURE[0].SIMPLE_DWORD := RETAINTEST_AUTO_ARRAYSIMPLESTRUCTURE[0].SIMPLE_DWORD + 1;
    RETAINTEST_AUTO_ARRAYSIMPLESTRUCTURE[0].SIMPLE_INT := RETAINTEST_AUTO_ARRAYSIMPLESTRUCTURE[0].SIMPLE_INT + 1;
    RETAINTEST_AUTO_ARRAYSIMPLESTRUCTURE[0].SIMPLE_LINT := RETAINTEST_AUTO_ARRAYSIMPLESTRUCTURE[0].SIMPLE_LINT + 1;
    RETAINTEST_AUTO_ARRAYSIMPLESTRUCTURE[0].SIMPLE_LREAL := RETAINTEST_AUTO_ARRAYSIMPLESTRUCTURE[0].SIMPLE_LREAL + 1.1;
    RETAINTEST_AUTO_ARRAYSIMPLESTRUCTURE[0].SIMPLE_LWORD := RETAINTEST_AUTO_ARRAYSIMPLESTRUCTURE[0].SIMPLE_LWORD + 1;
    RETAINTEST_AUTO_ARRAYSIMPLESTRUCTURE[0].SIMPLE_REAL := RETAINTEST_AUTO_ARRAYSIMPLESTRUCTURE[0].SIMPLE_REAL + 1.1;
    RETAINTEST_AUTO_ARRAYSIMPLESTRUCTURE[0].SIMPLE_SINT := RETAINTEST_AUTO_ARRAYSIMPLESTRUCTURE[0].SIMPLE_SINT + 1;
    RETAINTEST_AUTO_ARRAYSIMPLESTRUCTURE[0].SIMPLE_STRING := ANY_TO_STRING(RETAINTEST_AUTO_ARRAYSIMPLESTRUCTURE[0].SIMPLE_DINT) + ' ' + ANY_TO_STRING(RETAINTEST_AUTO_ARRAYSIMPLESTRUCTURE[0].SIMPLE_TIME);
    RETAINTEST_AUTO_ARRAYSIMPLESTRUCTURE[0].SIMPLE_TIME := RETAINTEST_AUTO_ARRAYSIMPLESTRUCTURE[0].SIMPLE_TIME + PULSE_TIME;
    RETAINTEST_AUTO_ARRAYSIMPLESTRUCTURE[0].SIMPLE_UDINT := RETAINTEST_AUTO_ARRAYSIMPLESTRUCTURE[0].SIMPLE_UDINT + 1;
    RETAINTEST_AUTO_ARRAYSIMPLESTRUCTURE[0].SIMPLE_UINT := RETAINTEST_AUTO_ARRAYSIMPLESTRUCTURE[0].SIMPLE_UINT + 1;
    RETAINTEST_AUTO_ARRAYSIMPLESTRUCTURE[0].SIMPLE_ULINT := RETAINTEST_AUTO_ARRAYSIMPLESTRUCTURE[0].SIMPLE_ULINT + 1;
    RETAINTEST_AUTO_ARRAYSIMPLESTRUCTURE[0].SIMPLE_USINT := RETAINTEST_AUTO_ARRAYSIMPLESTRUCTURE[0].SIMPLE_USINT + 1;
    RETAINTEST_AUTO_ARRAYSIMPLESTRUCTURE[0].SIMPLE_WORD := RETAINTEST_AUTO_ARRAYSIMPLESTRUCTURE[0].SIMPLE_WORD + 1;

    RETAINTEST_AUTO_ARRAYSIMPLESTRUCTURE[1].SIMPLE_BOOL := NOT RETAINTEST_AUTO_ARRAYSIMPLESTRUCTURE[1].SIMPLE_BOOL;
    RETAINTEST_AUTO_ARRAYSIMPLESTRUCTURE[1].SIMPLE_BYTE := RETAINTEST_AUTO_ARRAYSIMPLESTRUCTURE[1].SIMPLE_BYTE + 1;
    RETAINTEST_AUTO_ARRAYSIMPLESTRUCTURE[1].SIMPLE_DATE := ANY_TO_DATE(1445385600 + RETAINTEST_AUTO_ARRAYSIMPLESTRUCTURE[1].SIMPLE_DINT * 86400);
    RETAINTEST_AUTO_ARRAYSIMPLESTRUCTURE[1].SIMPLE_DINT := RETAINTEST_AUTO_ARRAYSIMPLESTRUCTURE[1].SIMPLE_DINT + 1;
    RETAINTEST_AUTO_ARRAYSIMPLESTRUCTURE[1].SIMPLE_DWORD := RETAINTEST_AUTO_ARRAYSIMPLESTRUCTURE[1].SIMPLE_DWORD + 1;
    RETAINTEST_AUTO_ARRAYSIMPLESTRUCTURE[1].SIMPLE_INT := RETAINTEST_AUTO_ARRAYSIMPLESTRUCTURE[1].SIMPLE_INT + 1;
    RETAINTEST_AUTO_ARRAYSIMPLESTRUCTURE[1].SIMPLE_LINT := RETAINTEST_AUTO_ARRAYSIMPLESTRUCTURE[1].SIMPLE_LINT + 1;
    RETAINTEST_AUTO_ARRAYSIMPLESTRUCTURE[1].SIMPLE_LREAL := RETAINTEST_AUTO_ARRAYSIMPLESTRUCTURE[1].SIMPLE_LREAL + 1.1;
    RETAINTEST_AUTO_ARRAYSIMPLESTRUCTURE[1].SIMPLE_LWORD := RETAINTEST_AUTO_ARRAYSIMPLESTRUCTURE[1].SIMPLE_LWORD + 1;
    RETAINTEST_AUTO_ARRAYSIMPLESTRUCTURE[1].SIMPLE_REAL := RETAINTEST_AUTO_ARRAYSIMPLESTRUCTURE[1].SIMPLE_REAL + 1.1;
    RETAINTEST_AUTO_ARRAYSIMPLESTRUCTURE[1].SIMPLE_SINT := RETAINTEST_AUTO_ARRAYSIMPLESTRUCTURE[1].SIMPLE_SINT + 1;
    RETAINTEST_AUTO_ARRAYSIMPLESTRUCTURE[1].SIMPLE_STRING := ANY_TO_STRING(RETAINTEST_AUTO_ARRAYSIMPLESTRUCTURE[1].SIMPLE_DINT) + ' ' + ANY_TO_STRING(RETAINTEST_AUTO_ARRAYSIMPLESTRUCTURE[1].SIMPLE_TIME);
    RETAINTEST_AUTO_ARRAYSIMPLESTRUCTURE[1].SIMPLE_TIME := RETAINTEST_AUTO_ARRAYSIMPLESTRUCTURE[1].SIMPLE_TIME + PULSE_TIME;
    RETAINTEST_AUTO_ARRAYSIMPLESTRUCTURE[1].SIMPLE_UDINT := RETAINTEST_AUTO_ARRAYSIMPLESTRUCTURE[1].SIMPLE_UDINT + 1;
    RETAINTEST_AUTO_ARRAYSIMPLESTRUCTURE[1].SIMPLE_UINT := RETAINTEST_AUTO_ARRAYSIMPLESTRUCTURE[1].SIMPLE_UINT + 1;
    RETAINTEST_AUTO_ARRAYSIMPLESTRUCTURE[1].SIMPLE_ULINT := RETAINTEST_AUTO_ARRAYSIMPLESTRUCTURE[1].SIMPLE_ULINT + 1;
    RETAINTEST_AUTO_ARRAYSIMPLESTRUCTURE[1].SIMPLE_USINT := RETAINTEST_AUTO_ARRAYSIMPLESTRUCTURE[1].SIMPLE_USINT + 1;
    RETAINTEST_AUTO_ARRAYSIMPLESTRUCTURE[1].SIMPLE_WORD := RETAINTEST_AUTO_ARRAYSIMPLESTRUCTURE[1].SIMPLE_WORD + 1;

    RETAINTEST_AUTO_ARRAYSIMPLESTRUCTURE[2].SIMPLE_BOOL := NOT RETAINTEST_AUTO_ARRAYSIMPLESTRUCTURE[2].SIMPLE_BOOL;
    RETAINTEST_AUTO_ARRAYSIMPLESTRUCTURE[2].SIMPLE_BYTE := RETAINTEST_AUTO_ARRAYSIMPLESTRUCTURE[2].SIMPLE_BYTE + 1;
    RETAINTEST_AUTO_ARRAYSIMPLESTRUCTURE[2].SIMPLE_DATE := ANY_TO_DATE(1445385600 + RETAINTEST_AUTO_ARRAYSIMPLESTRUCTURE[2].SIMPLE_DINT * 86400);
    RETAINTEST_AUTO_ARRAYSIMPLESTRUCTURE[2].SIMPLE_DINT := RETAINTEST_AUTO_ARRAYSIMPLESTRUCTURE[2].SIMPLE_DINT + 1;
    RETAINTEST_AUTO_ARRAYSIMPLESTRUCTURE[2].SIMPLE_DWORD := RETAINTEST_AUTO_ARRAYSIMPLESTRUCTURE[2].SIMPLE_DWORD + 1;
    RETAINTEST_AUTO_ARRAYSIMPLESTRUCTURE[2].SIMPLE_INT := RETAINTEST_AUTO_ARRAYSIMPLESTRUCTURE[2].SIMPLE_INT + 1;
    RETAINTEST_AUTO_ARRAYSIMPLESTRUCTURE[2].SIMPLE_LINT := RETAINTEST_AUTO_ARRAYSIMPLESTRUCTURE[2].SIMPLE_LINT + 1;
    RETAINTEST_AUTO_ARRAYSIMPLESTRUCTURE[2].SIMPLE_LREAL := RETAINTEST_AUTO_ARRAYSIMPLESTRUCTURE[2].SIMPLE_LREAL + 1.1;
    RETAINTEST_AUTO_ARRAYSIMPLESTRUCTURE[2].SIMPLE_LWORD := RETAINTEST_AUTO_ARRAYSIMPLESTRUCTURE[2].SIMPLE_LWORD + 1;
    RETAINTEST_AUTO_ARRAYSIMPLESTRUCTURE[2].SIMPLE_REAL := RETAINTEST_AUTO_ARRAYSIMPLESTRUCTURE[2].SIMPLE_REAL + 1.1;
    RETAINTEST_AUTO_ARRAYSIMPLESTRUCTURE[2].SIMPLE_SINT := RETAINTEST_AUTO_ARRAYSIMPLESTRUCTURE[2].SIMPLE_SINT + 1;
    RETAINTEST_AUTO_ARRAYSIMPLESTRUCTURE[2].SIMPLE_STRING := ANY_TO_STRING(RETAINTEST_AUTO_ARRAYSIMPLESTRUCTURE[2].SIMPLE_DINT) + ' ' + ANY_TO_STRING(RETAINTEST_AUTO_ARRAYSIMPLESTRUCTURE[2].SIMPLE_TIME);
    RETAINTEST_AUTO_ARRAYSIMPLESTRUCTURE[2].SIMPLE_TIME := RETAINTEST_AUTO_ARRAYSIMPLESTRUCTURE[2].SIMPLE_TIME + PULSE_TIME;
    RETAINTEST_AUTO_ARRAYSIMPLESTRUCTURE[2].SIMPLE_UDINT := RETAINTEST_AUTO_ARRAYSIMPLESTRUCTURE[2].SIMPLE_UDINT + 1;
    RETAINTEST_AUTO_ARRAYSIMPLESTRUCTURE[2].SIMPLE_UINT := RETAINTEST_AUTO_ARRAYSIMPLESTRUCTURE[2].SIMPLE_UINT + 1;
    RETAINTEST_AUTO_ARRAYSIMPLESTRUCTURE[2].SIMPLE_ULINT := RETAINTEST_AUTO_ARRAYSIMPLESTRUCTURE[2].SIMPLE_ULINT + 1;
    RETAINTEST_AUTO_ARRAYSIMPLESTRUCTURE[2].SIMPLE_USINT := RETAINTEST_AUTO_ARRAYSIMPLESTRUCTURE[2].SIMPLE_USINT + 1;
    RETAINTEST_AUTO_ARRAYSIMPLESTRUCTURE[2].SIMPLE_WORD := RETAINTEST_AUTO_ARRAYSIMPLESTRUCTURE[2].SIMPLE_WORD + 1;

    RETAINTEST_AUTO_ARRAYSIMPLESTRUCTURE[3].SIMPLE_BOOL := NOT RETAINTEST_AUTO_ARRAYSIMPLESTRUCTURE[3].SIMPLE_BOOL;
    RETAINTEST_AUTO_ARRAYSIMPLESTRUCTURE[3].SIMPLE_BYTE := RETAINTEST_AUTO_ARRAYSIMPLESTRUCTURE[3].SIMPLE_BYTE + 1;
    RETAINTEST_AUTO_ARRAYSIMPLESTRUCTURE[3].SIMPLE_DATE := ANY_TO_DATE(1445385600 + RETAINTEST_AUTO_ARRAYSIMPLESTRUCTURE[3].SIMPLE_DINT * 86400);
    RETAINTEST_AUTO_ARRAYSIMPLESTRUCTURE[3].SIMPLE_DINT := RETAINTEST_AUTO_ARRAYSIMPLESTRUCTURE[3].SIMPLE_DINT + 1;
    RETAINTEST_AUTO_ARRAYSIMPLESTRUCTURE[3].SIMPLE_DWORD := RETAINTEST_AUTO_ARRAYSIMPLESTRUCTURE[3].SIMPLE_DWORD + 1;
    RETAINTEST_AUTO_ARRAYSIMPLESTRUCTURE[3].SIMPLE_INT := RETAINTEST_AUTO_ARRAYSIMPLESTRUCTURE[3].SIMPLE_INT + 1;
    RETAINTEST_AUTO_ARRAYSIMPLESTRUCTURE[3].SIMPLE_LINT := RETAINTEST_AUTO_ARRAYSIMPLESTRUCTURE[3].SIMPLE_LINT + 1;
    RETAINTEST_AUTO_ARRAYSIMPLESTRUCTURE[3].SIMPLE_LREAL := RETAINTEST_AUTO_ARRAYSIMPLESTRUCTURE[3].SIMPLE_LREAL + 1.1;
    RETAINTEST_AUTO_ARRAYSIMPLESTRUCTURE[3].SIMPLE_LWORD := RETAINTEST_AUTO_ARRAYSIMPLESTRUCTURE[3].SIMPLE_LWORD + 1;
    RETAINTEST_AUTO_ARRAYSIMPLESTRUCTURE[3].SIMPLE_REAL := RETAINTEST_AUTO_ARRAYSIMPLESTRUCTURE[3].SIMPLE_REAL + 1.1;
    RETAINTEST_AUTO_ARRAYSIMPLESTRUCTURE[3].SIMPLE_SINT := RETAINTEST_AUTO_ARRAYSIMPLESTRUCTURE[3].SIMPLE_SINT + 1;
    RETAINTEST_AUTO_ARRAYSIMPLESTRUCTURE[3].SIMPLE_STRING := ANY_TO_STRING(RETAINTEST_AUTO_ARRAYSIMPLESTRUCTURE[3].SIMPLE_DINT) + ' ' + ANY_TO_STRING(RETAINTEST_AUTO_ARRAYSIMPLESTRUCTURE[3].SIMPLE_TIME);
    RETAINTEST_AUTO_ARRAYSIMPLESTRUCTURE[3].SIMPLE_TIME := RETAINTEST_AUTO_ARRAYSIMPLESTRUCTURE[3].SIMPLE_TIME + PULSE_TIME;
    RETAINTEST_AUTO_ARRAYSIMPLESTRUCTURE[3].SIMPLE_UDINT := RETAINTEST_AUTO_ARRAYSIMPLESTRUCTURE[3].SIMPLE_UDINT + 1;
    RETAINTEST_AUTO_ARRAYSIMPLESTRUCTURE[3].SIMPLE_UINT := RETAINTEST_AUTO_ARRAYSIMPLESTRUCTURE[3].SIMPLE_UINT + 1;
    RETAINTEST_AUTO_ARRAYSIMPLESTRUCTURE[3].SIMPLE_ULINT := RETAINTEST_AUTO_ARRAYSIMPLESTRUCTURE[3].SIMPLE_ULINT + 1;
    RETAINTEST_AUTO_ARRAYSIMPLESTRUCTURE[3].SIMPLE_USINT := RETAINTEST_AUTO_ARRAYSIMPLESTRUCTURE[3].SIMPLE_USINT + 1;
    RETAINTEST_AUTO_ARRAYSIMPLESTRUCTURE[3].SIMPLE_WORD := RETAINTEST_AUTO_ARRAYSIMPLESTRUCTURE[3].SIMPLE_WORD + 1;

    RETAINTEST_AUTO_ARRAYSIMPLESTRUCTURE[4].SIMPLE_BOOL := NOT RETAINTEST_AUTO_ARRAYSIMPLESTRUCTURE[4].SIMPLE_BOOL;
    RETAINTEST_AUTO_ARRAYSIMPLESTRUCTURE[4].SIMPLE_BYTE := RETAINTEST_AUTO_ARRAYSIMPLESTRUCTURE[4].SIMPLE_BYTE + 1;
    RETAINTEST_AUTO_ARRAYSIMPLESTRUCTURE[4].SIMPLE_DATE := ANY_TO_DATE(1445385600 + RETAINTEST_AUTO_ARRAYSIMPLESTRUCTURE[4].SIMPLE_DINT * 86400);
    RETAINTEST_AUTO_ARRAYSIMPLESTRUCTURE[4].SIMPLE_DINT := RETAINTEST_AUTO_ARRAYSIMPLESTRUCTURE[4].SIMPLE_DINT + 1;
    RETAINTEST_AUTO_ARRAYSIMPLESTRUCTURE[4].SIMPLE_DWORD := RETAINTEST_AUTO_ARRAYSIMPLESTRUCTURE[4].SIMPLE_DWORD + 1;
    RETAINTEST_AUTO_ARRAYSIMPLESTRUCTURE[4].SIMPLE_INT := RETAINTEST_AUTO_ARRAYSIMPLESTRUCTURE[4].SIMPLE_INT + 1;
    RETAINTEST_AUTO_ARRAYSIMPLESTRUCTURE[4].SIMPLE_LINT := RETAINTEST_AUTO_ARRAYSIMPLESTRUCTURE[4].SIMPLE_LINT + 1;
    RETAINTEST_AUTO_ARRAYSIMPLESTRUCTURE[4].SIMPLE_LREAL := RETAINTEST_AUTO_ARRAYSIMPLESTRUCTURE[4].SIMPLE_LREAL + 1.1;
    RETAINTEST_AUTO_ARRAYSIMPLESTRUCTURE[4].SIMPLE_LWORD := RETAINTEST_AUTO_ARRAYSIMPLESTRUCTURE[4].SIMPLE_LWORD + 1;
    RETAINTEST_AUTO_ARRAYSIMPLESTRUCTURE[4].SIMPLE_REAL := RETAINTEST_AUTO_ARRAYSIMPLESTRUCTURE[4].SIMPLE_REAL + 1.1;
    RETAINTEST_AUTO_ARRAYSIMPLESTRUCTURE[4].SIMPLE_SINT := RETAINTEST_AUTO_ARRAYSIMPLESTRUCTURE[4].SIMPLE_SINT + 1;
    RETAINTEST_AUTO_ARRAYSIMPLESTRUCTURE[4].SIMPLE_STRING := ANY_TO_STRING(RETAINTEST_AUTO_ARRAYSIMPLESTRUCTURE[4].SIMPLE_DINT) + ' ' + ANY_TO_STRING(RETAINTEST_AUTO_ARRAYSIMPLESTRUCTURE[4].SIMPLE_TIME);
    RETAINTEST_AUTO_ARRAYSIMPLESTRUCTURE[4].SIMPLE_TIME := RETAINTEST_AUTO_ARRAYSIMPLESTRUCTURE[4].SIMPLE_TIME + PULSE_TIME;
    RETAINTEST_AUTO_ARRAYSIMPLESTRUCTURE[4].SIMPLE_UDINT := RETAINTEST_AUTO_ARRAYSIMPLESTRUCTURE[4].SIMPLE_UDINT + 1;
    RETAINTEST_AUTO_ARRAYSIMPLESTRUCTURE[4].SIMPLE_UINT := RETAINTEST_AUTO_ARRAYSIMPLESTRUCTURE[4].SIMPLE_UINT + 1;
    RETAINTEST_AUTO_ARRAYSIMPLESTRUCTURE[4].SIMPLE_ULINT := RETAINTEST_AUTO_ARRAYSIMPLESTRUCTURE[4].SIMPLE_ULINT + 1;
    RETAINTEST_AUTO_ARRAYSIMPLESTRUCTURE[4].SIMPLE_USINT := RETAINTEST_AUTO_ARRAYSIMPLESTRUCTURE[4].SIMPLE_USINT + 1;
    RETAINTEST_AUTO_ARRAYSIMPLESTRUCTURE[4].SIMPLE_WORD := RETAINTEST_AUTO_ARRAYSIMPLESTRUCTURE[4].SIMPLE_WORD + 1;

    RETAINTEST_AUTO_ARRAYSIMPLESTRUCTURE[5].SIMPLE_BOOL := RETAINTEST_AUTO_ARRAYSIMPLESTRUCTURE[4].SIMPLE_BOOL;
    RETAINTEST_AUTO_ARRAYSIMPLESTRUCTURE[5].SIMPLE_BYTE := RETAINTEST_AUTO_ARRAYSIMPLESTRUCTURE[4].SIMPLE_BYTE;
    RETAINTEST_AUTO_ARRAYSIMPLESTRUCTURE[5].SIMPLE_DATE := RETAINTEST_AUTO_ARRAYSIMPLESTRUCTURE[4].SIMPLE_DATE;
    RETAINTEST_AUTO_ARRAYSIMPLESTRUCTURE[5].SIMPLE_DINT := RETAINTEST_AUTO_ARRAYSIMPLESTRUCTURE[4].SIMPLE_DINT;
    RETAINTEST_AUTO_ARRAYSIMPLESTRUCTURE[5].SIMPLE_DWORD := RETAINTEST_AUTO_ARRAYSIMPLESTRUCTURE[4].SIMPLE_DWORD;
    RETAINTEST_AUTO_ARRAYSIMPLESTRUCTURE[5].SIMPLE_INT := RETAINTEST_AUTO_ARRAYSIMPLESTRUCTURE[4].SIMPLE_INT;
    RETAINTEST_AUTO_ARRAYSIMPLESTRUCTURE[5].SIMPLE_LINT := RETAINTEST_AUTO_ARRAYSIMPLESTRUCTURE[4].SIMPLE_LINT;
    RETAINTEST_AUTO_ARRAYSIMPLESTRUCTURE[5].SIMPLE_LREAL := RETAINTEST_AUTO_ARRAYSIMPLESTRUCTURE[4].SIMPLE_LREAL;
    RETAINTEST_AUTO_ARRAYSIMPLESTRUCTURE[5].SIMPLE_LWORD := RETAINTEST_AUTO_ARRAYSIMPLESTRUCTURE[4].SIMPLE_LWORD;
    RETAINTEST_AUTO_ARRAYSIMPLESTRUCTURE[5].SIMPLE_REAL := RETAINTEST_AUTO_ARRAYSIMPLESTRUCTURE[4].SIMPLE_REAL;
    RETAINTEST_AUTO_ARRAYSIMPLESTRUCTURE[5].SIMPLE_SINT := RETAINTEST_AUTO_ARRAYSIMPLESTRUCTURE[4].SIMPLE_SINT;
    RETAINTEST_AUTO_ARRAYSIMPLESTRUCTURE[5].SIMPLE_STRING := RETAINTEST_AUTO_ARRAYSIMPLESTRUCTURE[4].SIMPLE_STRING;
    RETAINTEST_AUTO_ARRAYSIMPLESTRUCTURE[5].SIMPLE_TIME := RETAINTEST_AUTO_ARRAYSIMPLESTRUCTURE[4].SIMPLE_TIME;
    RETAINTEST_AUTO_ARRAYSIMPLESTRUCTURE[5].SIMPLE_UDINT := RETAINTEST_AUTO_ARRAYSIMPLESTRUCTURE[4].SIMPLE_UDINT;
    RETAINTEST_AUTO_ARRAYSIMPLESTRUCTURE[5].SIMPLE_UINT := RETAINTEST_AUTO_ARRAYSIMPLESTRUCTURE[4].SIMPLE_UINT;
    RETAINTEST_AUTO_ARRAYSIMPLESTRUCTURE[5].SIMPLE_ULINT := RETAINTEST_AUTO_ARRAYSIMPLESTRUCTURE[4].SIMPLE_ULINT;
    RETAINTEST_AUTO_ARRAYSIMPLESTRUCTURE[5].SIMPLE_USINT := RETAINTEST_AUTO_ARRAYSIMPLESTRUCTURE[4].SIMPLE_USINT;
    RETAINTEST_AUTO_ARRAYSIMPLESTRUCTURE[5].SIMPLE_WORD := RETAINTEST_AUTO_ARRAYSIMPLESTRUCTURE[4].SIMPLE_WORD;
END_IF;

END_PROGRAM
